(* CoDeSys 2.3 project: cy-12-wg-004.pro *)
(* Title: ClevergyAS - Albino E-02 *)
(* Version: 1.25 *)
(* Author: Andrea Ravasio *)
(* Libraries: Standard.lib 8.11.10 12:37:48, Util.lib 26.9.14 11:12:46, Visual.lib 8.11.10 12:37:48, Ethernet.lib 8.11.10 12:37:48, WagoLibIdent.lib 25.2.13 13:49:34, WagoLibMBX_01.lib 20.3.12 16:32:38, WagoLibStatus.lib 8.11.10 12:37:48, SysLibFile.lib 8.11.10 12:37:48, SysLibRtc.lib 8.11.10 12:37:48, SysLibSockets.lib 5.5.11 09:22:24, SysLibEvent.lib 8.11.10 12:37:48, SysLibPlcCtrl.lib 8.11.10 12:37:48, SysLibCallback.lib 8.11.10 12:37:48, ModbusEthernet_03.lib 15.5.15 16:47:39 *)

(* PLC configuration (modules and I/O channels)
VPN_ST1 AT %IX16.0 [BOOLOnX_I] Ch_1 Digital input
LAMP_AL AT %QX6.0 [BOOLOnX_Q] Ch_1 Digital output
KEY_QE_ST AT %IX16.1 [BOOLOnX_I] Ch_2 Digital input
CIR06_EN AT %QX6.1 [BOOLOnX_Q] Ch_2 Digital output
CIR07_AL AT %IX16.2 [BOOLOnX_I] Ch_3 Digital input
CIR05_EN AT %QX6.2 [BOOLOnX_Q] Ch_3 Digital output
CIR07_ST AT %IX16.3 [BOOLOnX_I] Ch_4 Digital input
CIR04_EN AT %QX6.3 [BOOLOnX_Q] Ch_4 Digital output
CIR07_AUT AT %IX16.4 [BOOLOnX_I] Ch_5 Digital input
CIR03_EN AT %QX6.4 [BOOLOnX_Q] Ch_5 Digital output
CIR06_AL AT %IX16.5 [BOOLOnX_I] Ch_6 Digital input
CIR02_EN AT %QX6.5 [BOOLOnX_Q] Ch_6 Digital output
CIR06_ST AT %IX16.6 [BOOLOnX_I] Ch_7 Digital input
CIR01_EN AT %QX6.6 [BOOLOnX_Q] Ch_7 Digital output
CIR06_AUT AT %IX16.7 [BOOLOnX_I] Ch_8 Digital input
CAL01_On_Off AT %QX6.7 [BOOLOnX_Q] Ch_8 Digital output
CIR05_AL AT %IX16.8 [BOOLOnX_I] Ch_1 Digital input
CIR07_EN AT %QX6.8 [BOOLOnX_Q] Ch_1 Digital output
CIR05_ST AT %IX16.9 [BOOLOnX_I] Ch_2 Digital input
CAL01_Rst_Bruc AT %QX6.9 [BOOLOnX_Q] Ch_2 Digital output
CIR05_AUT AT %IX16.10 [BOOLOnX_I] Ch_3 Digital input
AT %QX6.10 [BOOLOnX_Q] Ch_3 Digital output
CIR04_AL AT %IX16.11 [BOOLOnX_I] Ch_4 Digital input
AT %QX6.11 [BOOLOnX_Q] Ch_4 Digital output
CIR04_ST AT %IX16.12 [BOOLOnX_I] Ch_5 Digital input
AT %QX6.12 [BOOLOnX_Q] Ch_5 Digital output
CIR04_AUT AT %IX16.13 [BOOLOnX_I] Ch_6 Digital input
AT %QX6.13 [BOOLOnX_Q] Ch_6 Digital output
CIR03_AL AT %IX16.14 [BOOLOnX_I] Ch_7 Digital input
AT %QX6.14 [BOOLOnX_Q] Ch_7 Digital output
CIR03_ST AT %IX16.15 [BOOLOnX_I] Ch_8 Digital input
AT %QX6.15 [BOOLOnX_Q] Ch_8 Digital output
CIR03_AUT AT %IX17.0 [BOOLOnX_I] Ch_1 Digital input
CTL01_ST AT %IX17.1 [BOOLOnX_I] Ch_2 Digital input
CIR02_AUT AT %IX17.2 [BOOLOnX_I] Ch_3 Digital input
CIR01_AUT AT %IX17.3 [BOOLOnX_I] Ch_4 Digital input
ALARM_PM_PB_TB AT %IX17.4 [BOOLOnX_I] Ch_1 Digital input
CIR02_AL AT %IX17.5 [BOOLOnX_I] Ch_2 Digital input
UTA01_AL AT %IX17.6 [BOOLOnX_I] Ch_3 Digital input
CIR02_ST AT %IX17.7 [BOOLOnX_I] Ch_4 Digital input
CIR01_AL AT %IX17.8 [BOOLOnX_I] Ch_1 Digital input
CAL01_AL AT %IX17.9 [BOOLOnX_I] Ch_2 Digital input
CIR01_ST AT %IX17.10 [BOOLOnX_I] Ch_3 Digital input
CAL01_ManAuto AT %IX17.11 [BOOLOnX_I] Ch_4 Digital input
T_S01 AT %IW0 [INTOnW_I] Ch_1 signed Input value
T_S03 AT %IW1 [INTOnW_I] Ch_2 signed Input value
T_S02 AT %IW2 [INTOnW_I] Ch_3 signed Input value
T_S04 AT %IW3 [INTOnW_I] Ch_4 signed Input value
T_S05 AT %IW4 [INTOnW_I] Ch_1 signed Input value
T_S07 AT %IW5 [INTOnW_I] Ch_2 signed Input value
T_S06 AT %IW6 [INTOnW_I] Ch_3 signed Input value
AT %IW7 [INTOnW_I] Ch_4 signed Input value
T_S09 AT %IW8 [INTOnW_I] Ch_1 signed Input value
T_S08 AT %IW9 [INTOnW_I] Ch_2 signed Input value
AT %IW10 [INTOnW_I] Ch_3 signed Input value
AT %IW11 [INTOnW_I] Ch_4 signed Input value
VRD03_CTRL AT %QW0 [WORDOnW_Q] Ch_1 Analog output
VRD02_CTRL AT %QW1 [WORDOnW_Q] Ch_2 Analog output
VRD01_CTRL AT %QW2 [WORDOnW_Q] Ch_1 Analog output
VRD04_CTRL AT %QW3 [WORDOnW_Q] Ch_2 Analog output
CAL01_CRL AT %QW4 [WORDOnW_Q] Ch_1 Analog output
AT %QW5 [WORDOnW_Q] Ch_2 Analog output
VRD03_ST AT %IW12 [WORDOnW_I] Ch_1 Input word
VRD02_ST AT %IW13 [WORDOnW_I] Ch_2 Input word
0750-0478 2 AI 0-10V 16 Bit S.E. [Type_8_2_Channels] node 13, in %IB52 out %QB24 {INTTypePAAssignment = PLC; INTTypeModule = plugged}
  VRD01_ST AT %IW14 [WORDOnW_I] Ch_1 Input word
  VRD04_ST AT %IW15 [WORDOnW_I] Ch_2 Input word
0750-0513 2 DO 250V AC 2.0A Rel 2NO (PotFree) [Type_10_2_Channels] node 14, in %IB35 out %QB14 {INTTypePAAssignment = PLC; INTTypeModule = plugged}
  UTA_CTRL AT %QX7.0 [BOOLOnX_Q] Ch_1 Digital output
  AT %QX7.1 [BOOLOnX_Q] Ch_2 Digital output
Fieldbus variables [FB_VARS] node 1, in %IB0 out %QB0
Flag variables [FLAG_VARS] node 2, in %IB0 out %QB0
Modbus-Master [MB_MASTER] node 3, in %IB0 out %QB0
*)

(* Global variable list: Global_Constants *)
VAR_GLOBAL CONSTANT

	Plant_NAME			: STRING :='cySN:12 cyVER: E05 Palestra Centro Sportivo Rio Re ';
	Plant_SN			: DWORD  :=12;	(* S/N Impianto di telecontrollo *)
	Plant_SW_VER		: WORD   :=3;	(* Versione SW installata *)


	(* Parameters *)
	Plant_DefaultTAmb	: INT	:=100;		(* [.1°C] Temperatura ambiente di default in caso di rottura sonda *)
	Plant_MaxRunTAmb	: INT   :=250; 		(* [.1°C] Temperatura ambiente massima funzionamento impianto *)
	Plant_AntiFreezeTAmb: INT   :=-40;		(* [.1°C] Antifreeze temperature, start circulators *)
	Plant_CirOffDelay	: TIME	:=T#15m;	(* (Def.T#15m) Ritardo spegnimento pompe per ricircolo caldaia *)
	Plant_MaxWaterLoss	: WORD  :=2;		(* [lt/h] Massima perdita del circuito *)
	Plant_VRD_TDefault	: INT	:=300;		(* [.1°C] Temperatura di default in caso di errore climatica *)

	(* Filesystem *)
	FilesPath  			: STRING :='S:\';

(*	(* TCP Logger *)
	Logger_SERVER		: STRING:='';
	Logger_IP			: STRING:='192.168.100.3';
	Logger_PORT			: WORD  :=80;
	Logger_GETSTART		: STRING:='GET /cygmsrv/hsgm.ashx?';
	Logger_GETEND		: STRING:='$R$N$R$N';
	Logger_CHECK		: STRING:='True';
	Logger_CRLF			: STRING:='$R$N';
	Logger_DataFile		: STRING:='S:\LOG.DAT';
	Logger_DataFileOld	: STRING:='S:\LOG.BCK';
	Logger_IndexFile	: STRING:='S:\LOG.IDX';
	Logger_ConnRetries	: BYTE:=5;
	Logger_RecoverMsgs	: BYTE:=25;

	(* TCP Remote *)
	Remote_PORT			: WORD  :=10; (*44818; *)
	Remote_WELCOME		: STRING:='Connected$R$N';
	Remote_OK			: STRING:='OK$R$N';
	Remote_ERROR		: STRING:='ERROR$R$N';



	(* TCP Sockets *)
	MAX_SEND_TCP_SERVER					 : DWORD:=1500;(*60000*)
	MAX_RECEIVE_TCP_SERVER				 : DWORD:=3000;
	MAX_RECEIVE_TCP_SERVER_SOCKET	 	 : DWORD:=1500;
	MAX_SEND_TCP_CLIENT					 : DWORD:=3000;(*15000*)
	MAX_RECEIVE_TCP_CLIENT				 : DWORD:=1500;
	MAX_RECEIVE_TCP_CLIENT_SOCKET		 : DWORD:=1500;
	MAX_RECEIVE_UDP_SERVER				 : INT  :=1472;
	MAX_RECEIVE_UDP_CLIENT				 : INT  :=1472;
	CONNECT_WATCHDOG_TIME				 : TIME :=t#10s;
*)

	(* TCP Logger *)
	Logger_SERVER		: STRING:='';
	Logger_IP			: STRING:='192.168.100.3';
	Logger_PORT			: WORD  :=80;
	Logger_GETSTART		: STRING:='GET /cygmsrv/hsgm.ashx?';
	Logger_GETEND		: STRING:='$R$N$R$N';
	Logger_CHECK		: STRING:='True';
	Logger_CRLF			: STRING:='$R$N';
	Logger_DataFile		: STRING:='S:\LOG.DAT';
	Logger_DataFileOld	: STRING:='S:\LOG.BCK';
	Logger_IndexFile	: STRING:='S:\LOG.IDX';
	Logger_ConnRetries	: BYTE:=5;
	Logger_RecoverMsgs	: BYTE:=25;

	(* TCP Remote *)
	Remote_PORT			: WORD  :=10;
	Remote_WELCOME		: STRING:='Connected$R$N';
	Remote_OK			: STRING:='OK$R$N';
	Remote_ERROR		: STRING:='ERROR$R$N';

	(* TCP Sockets *)
	MAX_SEND_TCP_SERVER					 : DWORD:=3000;(*60000*)
	MAX_RECEIVE_TCP_SERVER				 : DWORD:=3000;
	MAX_RECEIVE_TCP_SERVER_SOCKET	 	 : DWORD:=1500;
	MAX_SEND_TCP_CLIENT					 : DWORD:=3000;(*15000*)
	MAX_RECEIVE_TCP_CLIENT				 : DWORD:=1500;
	MAX_RECEIVE_TCP_CLIENT_SOCKET		 : DWORD:=1500;
	MAX_RECEIVE_UDP_SERVER				 : INT  :=1472;
	MAX_RECEIVE_UDP_CLIENT				 : INT  :=1472;
	CONNECT_WATCHDOG_TIME				 : TIME :=t#10s;

	(* VISU COLORS *)
	COLOR_RED 			: DWORD:=16#2020F0;
	COLOR_YELLOW		: DWORD:=16#20F0F0;
	COLOR_GREEN			: DWORD:=16#20F020;
	COLOR_GREEN_OFF 	: DWORD:=16#006000;
	COLOR_LBLUE			: DWORD:=16#F0F080;
	COLOR_LIGHT_GREEN	: DWORD := 16#006000;





END_VAR

(* Global variable list: Global_Retain *)
VAR_GLOBAL RETAIN PERSISTENT
	CAL01_Clima : typ_Clima;
	VRD01_Clima : typ_Clima;
	VRD02_Clima : typ_Clima;
	VRD03_Clima : typ_Clima;
	VRD04_Clima : typ_Clima;

	CTL01_Count : DWORD;

	Mode_Manual : BOOL := FALSE;


	DelayAllarmeTemperaturaNonRaggiunta: INT;
	DeltaInterventoAllarmeTempeaturaNonRaggiuta: INT;
	OffsetSetPointManuale: INT;							(* Offset al Setpoint manuale per comensare lo scambiatore *)
	OffsetSetPointManuale2: INT;						(* Offset al Setpoint manuale per comensare lo scambiatore Aggiuntivo *)
	BitAbilitaBoost: BOOL:=TRUE;						(* Abilitiazione Boost *)
	RifOffsetBoost:INT;									(* Offset al Setpoint della Caldaia per azione di Boost *)

	SogliaMinStartAntigelo: INT;
	SogliaMinStopAntigelo: INT;
	BitAbilitaAntigelo: BOOL:=TRUE;


END_VAR

(* Global variable list: Global_Variables *)
VAR_GLOBAL

	SYS    : typ_SYS;
	Logger : typ_Logger;

	Lamp	:	LAMP_AL_GENERALE;

	T_AMB	:	INT;		(* Environment temperature *)


	(* Sonde Temperature impianto *)
	TPV01  : obj_TPV	:= ( ID:=1 ); 							   (* T_S01 Esterna *)
	TPV02  : obj_TPV	:= ( ID:=2 , IN_WMIN:=50 , IN_WMAX:=980 ); (* T_S02 Mandata Caldia *)
	TPV03  : obj_TPV	:= ( ID:=3 , IN_WMIN:=50 , IN_WMAX:=980 ); (* T_S03 Ritorno Caldaia *)
	TPV04  : obj_TPV	:= ( ID:=4 , IN_WMIN:=50 , IN_WMAX:=800 ); (* T_S04 FAN Coil Spogliatoio Piano Terra Radiatori*)
	TPV05  : obj_TPV	:= ( ID:=5 , IN_WMIN:=50 , IN_WMAX:=800 ); (* T_S05 Spogliatoio Primo Piano Radiatori *)
	TPV06  : obj_TPV	:= ( ID:=6 , IN_WMIN:=50 , IN_WMAX:=800 ); (* T_S06 Temperatura ACS *)
	TPV07  : obj_TPV	:= ( ID:=7 , IN_WMIN:=50 , IN_WMAX:=800 ); (* T_S07 Temperatura Bollitore *)
	TPV08  : obj_TPV	:= ( ID:=8 , IN_WMIN:=50 , IN_WMAX:=800 ); (* T_S08 Ingresso UTA *)
	TPV09  : obj_TPV	:= ( ID:=9 , IN_WMIN:=50 , IN_WMAX:=800 ); (* T_S09 Uscita UTA *)

	TAMB   : obj_TAMB	:= ( ID:=1 );
					(* vedi parametro G e Paramentro H manuale Caldaia UNICAL *)
	CAL01  : obj_CAL_01 := ( ID:=1,	LimiteMAXSetPoint:= 800,LimiteMinSetPoint:=300,OnDelay:=T#500ms,OffDelay:=T#500ms );


	(* Circolatori  *)
	CIR01  : obj_CIR_01 := ( ID:=1,CIR_AUTO:=TRUE, OnDelay:=T#1s, OffDelay:=T#5m);
	CIR02  : obj_CIR_01 := ( ID:=2,CIR_AUTO:=TRUE, OnDelay:=T#2s, OffDelay:=T#1s); (* Controllo Palestra UTA *)
	CIR03  : obj_CIR_01 := ( ID:=3,CIR_AUTO:=TRUE, OnDelay:=T#3s, OffDelay:=T#1s); (* Controllo Palestra Piano Terra Radiatori *)
	CIR04  : obj_CIR_01 := ( ID:=4,CIR_AUTO:=TRUE, OnDelay:=T#4s, OffDelay:=T#1s); (* Controllo Spogliatoi Primo Piano Radiatori *)
	CIR05  : obj_CIR_01 := ( ID:=5,CIR_AUTO:=TRUE, OnDelay:=T#5s, OffDelay:=T#1s); (* Controllo Circolatore Bollitore  *)
	CIR06  : obj_CIR_01 := ( ID:=6,CIR_AUTO:=TRUE, OnDelay:=T#6s, OffDelay:=T#1s); (* Controllo Circolatore Bollitore  *)
	CIR07  : obj_CIR_01 := ( ID:=7,CIR_AUTO:=TRUE, OnDelay:=T#7s, OffDelay:=T#1s); (* Controllo Circolatore ACS *)


	(* Valvole motorizzate Analogiche  *)
	VRD01	:	obj_VRD_02:= (ID:=1, fFeedback:=TRUE, ReducedRange := FALSE,Local_VRD_TAlarm:=800); (* Controllo Palestra Piano Terra Radiatori *)
	VRD02	:	obj_VRD_02:= (ID:=2, fFeedback:=TRUE, ReducedRange := FALSE,Local_VRD_TAlarm:=800); (* Controllo Spogliatoi Primo Piano Radiatori *)
(* VRD03 Esclusa perchè bypassata *)
(*	VRD03	:	obj_VRD_02:= (ID:=3, fFeedback:=TRUE, ReducedRange := FALSE,Local_VRD_TAlarm:=800); (* Controllo Circolatore Bollitore  *) *)
	VRD04	:	obj_VRD_02:= (ID:=4, fFeedback:=TRUE, ReducedRange := FALSE,Local_VRD_TAlarm:=800); (* Controllo Palestra UTA *)


	(* Crono termostati *)
	THER01 : obj_CRONTER := ( ID:=1, Local_MaxRunTAmb:=800,Histeresys:=10); (* Controllo Palestra UTA *)
	THER02 : obj_CRONTER := ( ID:=2, Local_MaxRunTAmb:=800,Histeresys:=10);	(* Controllo Palestra Piano Terra Radiatori *)
	THER03 : obj_CRONTER := ( ID:=3, Local_MaxRunTAmb:=800,Histeresys:=10);	(* Controllo Spogliatoi Primo Piano Radiatori *)
	THER04 : obj_CRONTER := ( ID:=4, Local_MaxRunTAmb:=800,Histeresys:=50);	(* Controllo Circolatore Bollitore  *)
	THER05 : obj_CRONTER := ( ID:=5, Local_MaxRunTAmb:=800,Histeresys:=10);	(* Controllo Circolatore ACS *)
	THER250: obj_CRONTER := ( ID:=250, Local_MaxRunTAmb:=800,Histeresys:=10);(* Controllo Boost *)

	CronEd : obj_CRON_EDITOR;

	(* Contalitri *)
	CTL01	:	obj_CTL	:= (ID:=1, Peso:=10);
	UTA01  : obj_UTA:=(ID:=1);



	UTA01_ST: BOOL;
	UTA01_Antigelo: BOOL;
	UTA01_ManAut: BOOL;
END_VAR

(* Data type in LON/Enumerations *)
TYPE alarm_type_t :
(
	AL_HEADER := -13,
	AL_FOOTER := -12,
	AL_DEBUG := -11,
	AL_INFO := -10,
	AL_SYSTEM_INFO := -6,
	AL_VALUE_INVALID := -5,
	AL_CONSTANT := -4,
	AL_OFFLINE := -3,
	AL_UNKNOWN := -2,
	AL_NUL := -1,
	AL_NO_CONDITION := 0,
	AL_ALM_CONDITION := 1,
	AL_TOT_SVC_ALM_1 := 2,
	AL_TOT_SVC_ALM_2 := 3,
	AL_TOT_SVC_ALM_3 := 4,
	AL_LOW_LMT_CLR_1 := 5,
	AL_LOW_LMT_CLR_2 := 6,
	AL_HIGH_LMT_CLR_1 := 7,
	AL_HIGH_LMT_CLR_2 := 8,
	AL_LOW_LMT_ALM_1 := 9,
	AL_LOW_LMT_ALM_2 := 10,
	AL_HIGH_LMT_ALM_1 := 11,
	AL_HIGH_LMT_ALM_2 := 12,
	AL_FIR_ALM := 13,
	AL_FIR_PRE_ALM := 14,
	AL_FIR_TRBL := 15,
	AL_FIR_SUPV := 16,
	AL_FIR_TEST_ALM := 17,
	AL_FIR_TEST_PRE_ALM := 18,
	AL_FIR_ENVCOMP_MAX := 19,
	AL_FIR_MONITOR_COND := 20,
	AL_FIR_MAINT_ALERT := 21,
	AL_FATAL_ERROR := 30,
	AL_ERROR := 31,
	AL_WARNING := 32
);
END_TYPE

(* Data type in Errors *)
TYPE en_Logger_ErrLev :
(
	EL_Log			:=0,
	EL_Wrn			:=1,
	EL_Alarm		:=2,
	EL_AlarmStop	:=3
);
END_TYPE

(* Data type in Errors *)
TYPE en_Logger_Status :
(
	S_Logger_UNKNOWN := 0,
	S_Logger_IDLE,
	S_Logger_WAITCONN,
	S_Logger_WAITTX,
	S_Logger_WAITRESP,
	S_Logger_ERROR
);
END_TYPE

(* Data type *)
TYPE en_SYS_Objects :
(
	EO_SYS		:=0,  (* PLC *)
	EO_VPN		:=1,  (* VPN *)
	EO_DOOR		:=2,  (* Door & access control *)

	EO_CAL		:=10, (* Caldaia *)
	EO_CIR		:=11, (* Circolatore *)
	EO_CRON		:=12, (* Crono-termostato *)
	EO_VRD		:=13, (* Valvola miscelatore pannelli *)
	EO_CTL		:=14, (* Contalitri *)
	EO_CTB		:=15, (* Contabilizzatore *)
	EO_TPV		:=16, (* Temperature probes values *)
	EO_PPV		:=17, (* Pressure probes values *)
	EO_PBV		:=18, (* Over-Pressure Alarms *)
	EO_TBV		:=19, (* Over-Temperature Alarms *)
	EO_PMV		:=20, (* Under-Pressure Alarms *)
	EO_GRU		:=21, (* Gruppo termico *)
	EO_PDC		:=22, (* Pompa di calore *)
	EO_SOL		:=23, (* Pannello solare termico *)
	EO_ESOL		:=24, (* Pannello solare fotovoltaico *)
	EO_GAS		:=25, (* Contatore GAS *)
	EO_PORT		:=26, (* Misuratore di portata *)
	EO_FPV		:=27, (* Flow probes values *)
	EO_ANZ		:=28, (* Analizzatore di rete *)
	EO_SCA		:=29, (* Signal Control Alarms *)
	EO_LUX		:=30, (* Base Illumination point *)
	EO_LUXM		:=31, (* Metered Illumination point *)
	EO_PSG		:=32, (* Sensore di passaggio *)
	EO_HVAC		:=33, (* Heating, Ventilating and Air Conditioning *)
	EO_HYGRV	:=34, (* Relative Humidity sensors value *)
	EO_COOV		:=35, (* Carbon Dioxide CO2 sensors value *)
	EO_INV		:=36, (* Inverter *)
	EO_STR		:=37, (* Smart string box *)

	EO_CIRD		:=39, (* Double CIR *)
	EO_ACS		:=40, (* Hot domestic water *)
	EO_FRG		:=41, (* Frigo *)
	EO_THER		:=42, (* Thermostat *)
	EO_CIRM		:=43, (* Modbus CIR *)
	EO_CIRDM	:=44, (* Modbus double CIR *)
	EO_UTA		:=47, (* Modbus double CIR *)

	EO_ZGW			:=200,  (* ZigBee - Gateway *)
	EO_ZRM			:=201,	(* ZigBee - Repeater *)
	EO_ZREL			:=202,	(* ZigBee - Actuator rele *)
	EO_ZTHL			:=203,	(* ZigBee - Temperature Sensor *)

	EO_ASGW			:=250,	(* ASi - Gateway *)
	EO_ASCBI		:=251,	(* ASi - Input Board, Ciabatta *)

	EO_LON			:=1000, (* Bus - LON *)
	EO_MODBUS		:=1001, (* Bus - MODBUS *)
	EO_MBUS			:=1002, (* Bus - M-BUS *)
	EO_MODBUS_TCP	:=1003, (* Bus - MODBUS TCP *)

	EO_GENERIC		:=9000, (* Generic dataset *)
	EO_EXPO			:=9001 (* EXPO dataset *)
);
END_TYPE

(* Data type *)
TYPE en_SYS_Status :
(
	S_UNKNOWN  := 0,
	S_STARTUP,
	S_INIT_RTC,
	S_INIT_VAR,
	S_AUTOTEST,
	S_RUNNING,
	S_SHUTDOWN,
	S_HALT
);
END_TYPE

(* Data type in LON/Enumerations *)
TYPE file_request_t :
(
	FR_NUL := -1,
	FR_OPEN_TO_SEND := 0,
	FR_OPEN_TO_RECEIVE := 1,
	FR_CLOSE_FILE := 2,
	FR_CLOSE_DELETE_FILE := 3,
	FR_DIRECTORY_LOOKUP := 4,
	FR_OPEN_TO_SEND_RA := 5,
	FR_OPEN_TO_RECEIVE_RA := 6
);
END_TYPE

(* Data type in LON/Enumerations *)
TYPE file_status_t :
(
	FS_NUL := -1,
	FS_XFER_OK := 0,
	FS_LOOKUP_OK := 1,
	FS_OPEN_FAIL := 2,
	FS_LOOKUP_ERR := 3,
	FS_XFER_UNDERWAY := 4,
	FS_IO_ERR := 5,
	FS_TIMEOUT_ERR := 6,
	FS_WINDOW_ERR := 7,
	FS_AUTH_ERR := 8,
	FS_ACCESS_UNAVAIL := 9,
	FS_SEEK_INVALID := 10,
	FS_SEEK_WAIT := 11
);
END_TYPE

(* Data type in LON/Enumerations *)
TYPE hvac_t :
(
	HVAC_NUL := -1,
	HVAC_AUTO := 0,
	HVAC_HEAT := 1,
	HVAC_MRNG_WRMUP := 2,
	HVAC_COOL := 3,
	HVAC_NIGHT_PURGE := 4,
	HVAC_PRE_COOL := 5,
	HVAC_OFF := 6,
	HVAC_TEST := 7,
	HVAC_EMERG_HEAT := 8,
	HVAC_FAN_ONLY := 9,
	HVAC_FREE_COOL := 10,
	HVAC_ICE := 11,
	HVAC_MAX_HEAT := 12,
	HVAC_ECONOMY := 13,
	HVAC_DEHUMID := 14,
	HVAC_CALIBRATE := 15,
	HVAC_EMERG_COOL := 16,
	HVAC_EMERG_STEAM := 17,
	HVAC_MAX_COOL := 18,
	HVAC_HVC_LOAD := 19,
	HVAC_NO_LOAD := 20
);
END_TYPE

(* Data type in LON/Enumerations *)
TYPE object_request_t :
(
	RQ_NUL := -1,
	RQ_NORMAL := 0,
	RQ_DISABLED := 1,
	RQ_UPDATE_STATUS := 2,
	RQ_SELF_TEST := 3,
	RQ_UPDATE_ALARM := 4,
	RQ_REPORT_MASK := 5,
	RQ_OVERRIDE := 6,
	RQ_ENABLE := 7,
	RQ_RMV_OVERRIDE := 8,
	RQ_CLEAR_STATUS := 9,
	RQ_CLEAR_ALARM := 10,
	RQ_ALARM_NOTIFY_ENABLED := 11,
	RQ_ALARM_NOTIFY_DISABLED := 12,
	RQ_MANUAL_CTRL := 13,
	RQ_REMOTE_CTRL := 14,
	RQ_PROGRAM := 15,
	RQ_CLEAR_RESET := 16,
	RQ_RESET := 17,
	RQ_CLEAR_LOG := 18,
	RQ_LOAD_PROGRAM := 19,
	RQ_RUN_PROGRAM := 20,
	RQ_HALT_PROGRAM := 21,
	RQ_RESTART_PROGRAM := 22,
	RQ_UNLOAD_PROGRAM := 23,
	RQ_STEP_PROGRAM := 24
);
END_TYPE

(* Data type in LON/Enumerations *)
TYPE priority_level_t :
(
	PR_NUL := -1,
	PR_LEVEL_0 := 0,
	PR_LEVEL_1 := 1,
	PR_LEVEL_2 := 2,
	PR_LEVEL_3 := 3,
	PR_1 := 4,
	PR_2 := 5,
	PR_3 := 6,
	PR_4 := 7,
	PR_6 := 8,
	PR_8 := 9,
	PR_10 := 10,
	PR_16 := 11
);
END_TYPE

(* Data type in Plant_Objects *)
TYPE typ_Clima : (* CURVA CLIMATICA *)
STRUCT
	InitOK:		BOOL;
	Points: 	ARRAY [0..10] OF POINT;
END_STRUCT
END_TYPE

(* Data type in Plant_Objects *)
TYPE typ_Cron_Calendar :
STRUCT
	Profile		: ARRAY[0..384] OF BYTE;
END_STRUCT
END_TYPE

(* Data type in Plant_Objects *)
TYPE typ_Cron_Jolly :
STRUCT
	Start		: DT;
	End			: DT;
	Temp		: WORD;
	Flags		: WORD; (* B0:Enabled B1..B15:Unused *)
END_STRUCT
END_TYPE

(* Data type in Plant_Objects *)
TYPE typ_Cron_Profile :
STRUCT
	Flags		: WORD;
	Setpoint	: ARRAY [0..95] OF WORD;
END_STRUCT
END_TYPE

(* Data type in Errors *)
TYPE typ_Logger :
STRUCT
	Status		: en_Logger_Status;

	SendReq		: BOOL;
	SendIdx		: DWORD;
	SendData	: ARRAY [0..MAX_SEND_TCP_CLIENT] OF BYTE;
	SendLen		: DINT;

	TData		: ARRAY [0..MAX_SEND_TCP_CLIENT] OF BYTE;
	TLen		: DINT;

	LastIdxPos	: DWORD;

	(* Temporary variables used by objects *)
	s1			: STRING(256);
	i1			: WORD;


END_STRUCT
END_TYPE

(* Data type in Plant_Objects *)
TYPE typ_MODBUS_VAR : (* Gestione parametri MODBUS *)
STRUCT
	SlaveAddress	: BYTE;
	FunCode			: BYTE;
	FunAddress		: WORD;
	Refresh_Time	: BYTE; (* 0:No refresh x:Refresh in seconds *)
	Refresh_Cnt		: BYTE; (* INTERNAL *)
	Variable		: POINTER TO WORD;
	Variable_Size	: BYTE;
	Variable_Mirror : WORD; (* INTERNAL [Force refresh on read variables when <>0] *)
END_STRUCT
END_TYPE

(* Data type *)
TYPE typ_SYS :
STRUCT
	Status			: en_SYS_Status;
	Warning			: BOOL;
	Alarm			: BOOL;
	AlarmStop		: BOOL;

	Time_LogString	: STRING;
	Time_Year		: WORD;
	Time_Month		: BYTE;
	Time_Day		: BYTE;

	Time_CT_DT		: DT;
	Time_CT_Day		: WORD;
	Time_CT_Quarter	: BYTE;

	LastLogs_Idx	: BYTE;
	LastLogs_Dat	: ARRAY[0..5] OF STRING;
	LastLogs_Msg	: ARRAY[0..5] OF STRING;

END_STRUCT
END_TYPE

(* Data type in LON/NetworkVariables *)
TYPE typSnvtAlarm : 
STRUCT
	abLocation : ARRAY[0..5] OF BYTE;
	wObjectId : WORD;
	bAlarmType : BYTE (* enum type alarm_type_t *);
	bPriorityLevel : BYTE (* enum type priority_level_t *);
	wIndexToSnvt : WORD;
	abValue : ARRAY[0..3] OF BYTE;
	wYear : WORD;
	bMonth : BYTE;
	bDay : BYTE;
	bHour : BYTE;
	bMinute : BYTE;
	bSecond : BYTE;
	wMillisecond : WORD;
	abAlarmLimit : ARRAY[0..3] OF BYTE;
	bStatusInformation : BYTE; (* bit allocation of bStatusInformation:
	bit 0: NVI update counter LSB
	bit 1: NVI update counter
	bit 2: NVI update counter
	bit 3: NVI update counter MSB
	bit 4: timeout for NVI occurs (MaxRcvTime expired)
	bit 5: reserved
	bit 6: reserved
	bit 7: force NVO update *)
	bInternalUseOnly : BYTE; (* Do not use this byte in your application! *)
END_STRUCT
END_TYPE

(* Data type in LON/NetworkVariables *)
TYPE typSnvtFilePos : 
STRUCT
	diRwPtr : DINT;
	wRwLength : WORD;
	bStatusInformation : BYTE; (* bit allocation of bStatusInformation:
	bit 0: NVI update counter LSB
	bit 1: NVI update counter
	bit 2: NVI update counter
	bit 3: NVI update counter MSB
	bit 4: timeout for NVI occurs (MaxRcvTime expired)
	bit 5: reserved
	bit 6: reserved
	bit 7: force NVO update *)
	bInternalUseOnly : BYTE; (* Do not use this byte in your application! *)
END_STRUCT
END_TYPE

(* Data type in LON/NetworkVariables *)
TYPE typSnvtFileReq : 
STRUCT
	bRequest : BYTE (* enum type file_request_t *);
	wIndex : WORD;
	wReceiveTimeout : WORD;
	abDestAddress : ARRAY[0..4] OF BYTE (* union declaration *);
	bAuthOn : BYTE;
	bPrioOn : BYTE;
	bStatusInformation : BYTE; (* bit allocation of bStatusInformation:
	bit 0: NVI update counter LSB
	bit 1: NVI update counter
	bit 2: NVI update counter
	bit 3: NVI update counter MSB
	bit 4: timeout for NVI occurs (MaxRcvTime expired)
	bit 5: reserved
	bit 6: reserved
	bit 7: force NVO update *)
	bInternalUseOnly : BYTE; (* Do not use this byte in your application! *)
END_STRUCT
END_TYPE

(* Data type in LON/NetworkVariables *)
TYPE typSnvtFileStatus : 
STRUCT
	bStatus : BYTE (* enum type file_status_t *);
	wNumberOfFiles : WORD;
	wSelectedFile : WORD;
	abAdr : ARRAY[0..21] OF BYTE (* union declaration *);
	bStatusInformation : BYTE; (* bit allocation of bStatusInformation:
	bit 0: NVI update counter LSB
	bit 1: NVI update counter
	bit 2: NVI update counter
	bit 3: NVI update counter MSB
	bit 4: timeout for NVI occurs (MaxRcvTime expired)
	bit 5: reserved
	bit 6: reserved
	bit 7: force NVO update *)
	bInternalUseOnly : BYTE; (* Do not use this byte in your application! *)
END_STRUCT
END_TYPE

(* Data type in LON/NetworkVariables *)
TYPE typSnvtHvacMode : 
STRUCT
	bSnvtHvacMode : BYTE (* enum type hvac_t *);
	bStatusInformation : BYTE; (* bit allocation of bStatusInformation:
	bit 0: NVI update counter LSB
	bit 1: NVI update counter
	bit 2: NVI update counter
	bit 3: NVI update counter MSB
	bit 4: timeout for NVI occurs (MaxRcvTime expired)
	bit 5: reserved
	bit 6: reserved
	bit 7: force NVO update *)
	bInternalUseOnly : BYTE; (* Do not use this byte in your application! *)
END_STRUCT
END_TYPE

(* Data type in LON/NetworkVariables *)
TYPE typSnvtObjRequest : 
STRUCT
	wObjectId : WORD;
	bObjectRequest : BYTE (* enum type object_request_t *);
	bStatusInformation : BYTE; (* bit allocation of bStatusInformation:
	bit 0: NVI update counter LSB
	bit 1: NVI update counter
	bit 2: NVI update counter
	bit 3: NVI update counter MSB
	bit 4: timeout for NVI occurs (MaxRcvTime expired)
	bit 5: reserved
	bit 6: reserved
	bit 7: force NVO update *)
	bInternalUseOnly : BYTE; (* Do not use this byte in your application! *)
END_STRUCT
END_TYPE

(* Data type in LON/NetworkVariables *)
TYPE typSnvtObjStatus : 
STRUCT
	wObjectId : WORD;
	bBitfieldByteOffset2 : BYTE (* bit field *);
	bBitfieldByteOffset3 : BYTE (* bit field *);
	bBitfieldByteOffset4 : BYTE (* bit field *);
	bBitfieldByteOffset5 : BYTE (* bit field *);
	bStatusInformation : BYTE; (* bit allocation of bStatusInformation:
	bit 0: NVI update counter LSB
	bit 1: NVI update counter
	bit 2: NVI update counter
	bit 3: NVI update counter MSB
	bit 4: timeout for NVI occurs (MaxRcvTime expired)
	bit 5: reserved
	bit 6: reserved
	bit 7: force NVO update *)
	bInternalUseOnly : BYTE; (* Do not use this byte in your application! *)
END_STRUCT
END_TYPE

(* Data type in LON/NetworkVariables *)
TYPE typSnvtState : 
STRUCT
	bBitfieldByteOffset0 : BYTE (* bit field *);
	bBitfieldByteOffset1 : BYTE (* bit field *);
	bStatusInformation : BYTE; (* bit allocation of bStatusInformation:
	bit 0: NVI update counter LSB
	bit 1: NVI update counter
	bit 2: NVI update counter
	bit 3: NVI update counter MSB
	bit 4: timeout for NVI occurs (MaxRcvTime expired)
	bit 5: reserved
	bit 6: reserved
	bit 7: force NVO update *)
	bInternalUseOnly : BYTE; (* Do not use this byte in your application! *)
END_STRUCT
END_TYPE

(* Data type in LON/NetworkVariables *)
TYPE typSnvtSwitch : 
STRUCT
	bValue : BYTE;
	siState : SINT;
	bStatusInformation : BYTE; (* bit allocation of bStatusInformation:
	bit 0: NVI update counter LSB
	bit 1: NVI update counter
	bit 2: NVI update counter
	bit 3: NVI update counter MSB
	bit 4: timeout for NVI occurs (MaxRcvTime expired)
	bit 5: reserved
	bit 6: reserved
	bit 7: force NVO update *)
	bInternalUseOnly : BYTE; (* Do not use this byte in your application! *)
END_STRUCT
END_TYPE

(* Data type in LON/NetworkVariables *)
TYPE typSnvtTempP :
STRUCT
	iSnvtTempP : INT;
	bStatusInformation : BYTE; (* bit allocation of bStatusInformation:
	bit 0: NVI update counter LSB
	bit 1: NVI update counter
	bit 2: NVI update counter
	bit 3: NVI update counter MSB
	bit 4: timeout for NVI occurs (MaxRcvTime expired)
	bit 5: reserved
	bit 6: reserved
	bit 7: force NVO update *)
	bInternalUseOnly : BYTE; (* Do not use this byte in your application! *)
END_STRUCT
END_TYPE

(* Data type in LON/NetworkVariables *)
TYPE typSnvtTimeStamp : 
STRUCT
	iYear : INT;
	bMonth : BYTE;
	bDay : BYTE;
	bHour : BYTE;
	bMinute : BYTE;
	bSecond : BYTE;
	bStatusInformation : BYTE; (* bit allocation of bStatusInformation:
	bit 0: NVI update counter LSB
	bit 1: NVI update counter
	bit 2: NVI update counter
	bit 3: NVI update counter MSB
	bit 4: timeout for NVI occurs (MaxRcvTime expired)
	bit 5: reserved
	bit 6: reserved
	bit 7: force NVO update *)
	bInternalUseOnly : BYTE; (* Do not use this byte in your application! *)
END_STRUCT
END_TYPE

(* POU PLC_PRG, ST *)
PROGRAM PLC_PRG
VAR
	Timer1: TON; (* Fast controls tick *)
	Timer2: TON; (* Plant control tick *)
	Timer3: TON; (* Logger timer *)

	SecCircuitLogic	:	BOOL;	(* Secondary circuit request: LOGICAL ON/OFF *)
	SecCircuitReal	:	BOOL;	(* Secondart circuit request: REAL ON/OFF	 *)




	StartCAL_Antigelo: RS;
	fAntigelo		:FLT_TAP;  (* Sgnalazione LOG Antigelo  *)


	OffsetBoost: INT;
	pippo: WORD;
	HMI_AggiornaLog: BOOL;
	SetPointVRD04: INT;

	OffsetVRD04: INT;

END_VAR

VAR RETAIN
	HMISetPointVRD04: INT;
	HMI_LimitMaxOut: INT;
	HMI_LimitMinOut:INT;
	HMI_LimitMinIN: INT;
	HMI_LimitMaxIN: INT;
END_VAR
(******************************************************************************
 ****                           MAIN TASK CODE                             ****
 ******************************************************************************

	Network setup:
		IP  = 192.168.100.2 | MSK = 255.255.255.0
		GW	= 192.168.100.1 | DNS = 192.168.100.1
		SNTP = 193.204.114.232 (3600s) ==> 192.168.100.3
*)

(*==============================*)
(*===== Main status machine ====*)
(*==============================*)
Main_Stm();

(*==============================*)
(*== Running cycle operations ==*)
(*==============================*)
(*
IF SYS.Status>S_INIT_VAR THEN

	(* Update LON output variables (needs to be here to obtain only one refresh) *)
	CAL01.Heartbeat( CLIM:=CAL01_Clima );
	(* Execute LON process *)
	Module_1_PRG();

END_IF
*)
(*==============================*)
(*== System cycle operations ===*)
(*==============================*)
(* Execute TCP processes *)
Logger_Proc();
Remote_Proc();
(* Update user led *)
USRLED_Update();
(* Execute Cron Editor commands *)
CronEd();
END_PROGRAM
ACTION Main_Stm:
CASE Sys.Status OF

	S_STARTUP:
		Sys.Status:=S_INIT_RTC;

	S_INIT_RTC:
		(* Check RTC and update from network *)
		RTC_Update();
		(* Check time *)
		IF Sys.Time_Year>2000 THEN
			Sys.Status:=S_INIT_VAR;
		END_IF








	S_INIT_VAR:
		LogEv(EL_Wrn,EO_SYS,0,1,CONCAT('System_startup_v',WORD_TO_STRING(Plant_SW_VER)));
		Sys.Status:=S_RUNNING;

	S_RUNNING:
		Timer1(IN:=NOT Timer1.Q,PT:=T#50ms);
		IF Timer1.Q THEN
			(* Update meters *)
			CTL01 ( CTL_ST:=CTL01_ST, COUNT:=CTL01_Count );
			(* Update system checks *)
			SYS_Proc();
		END_IF

		Timer2(IN:=NOT Timer2.Q,PT:=T#500ms);
		IF Timer2.Q THEN
			(* Read current date/time *)
			RTC_Update();
			(* Execute plant operations *)
			TPV01	 ( IN:=T_S01);
			TPV02	 ( IN:=T_S02);
			TPV03	 ( IN:=T_S03);
			TPV04	 ( IN:=T_S04);
			TPV05	 ( IN:=T_S05);
			TPV06	 ( IN:=T_S06);
			TPV07	 ( IN:=T_S07);
			TPV08	 ( IN:=T_S08);
			TPV09	 ( IN:=T_S09);

		(*	TAMB  ( IN1:=TPV01.IN ); *)
			T_AMB:=TPV01.IN;

			(* Crono, CronoTermostati e boost ed eventuale Antigelo  *)

(*
		  (* Gestione Ciclo antigelo : in questo impianto il ciclo antigelo è gestito coi crono ambiente *)

			StartCAL_Antigelo(	SET:=(SogliaMinStartAntigelo>TPV03.AVG),
								RESET1:= (TPV03.AVG>SogliaMinStopAntigelo) OR NOT BitAbilitaAntigelo
							);



			fAntigelo(IN:=StartCAL_Antigelo.Q1);
			IF fAntigelo.EVH THEN
				LogEv(EL_Log,EO_SYS,0,11,'Ciclo_Antigelo_Attivato');
			END_IF
			IF fAntigelo.EVL THEN
				LogEv(EL_Log,EO_SYS,0,12,'Ciclo_Antigelo_Disattivato');
			END_IF
*)



			THER01();						(* gestito solo Crono *)
			CIR02.OnOff:=THER01.RunCrono; 	(* UTA Palestra Fan Coil *) (* OR StartCAL_Antigelo.Q1 -- per introdurre start antigelo *)

			THER02();						(* gestito solo Crono *)
			CIR03.OnOff:=THER02.RunCrono; 	(* Spogliatoio Piano Terra Radiatori *)

			THER03();						(* gestito solo Crono *)
			CIR04.OnOff:=THER03.RunCrono; 	(* Spgliatoio Piano Primo Radiatori *)

			THER04(Temperature:=TPV07.IN);				(* gestito solo Cronotermostato *)
			CIR05.OnOff:=CIR06.OnOff:=THER04.Run; 	(* Bollitore *)

			THER05();						(* gestito solo Crono *)
			CIR07.OnOff:=THER05.RunCrono; 	(* Lancio ACS *)

			(* il crono virtuale 250 è quello che gestisce il boost.
				 Questo è attivo se da remoto lo abilitano ed è subordinato alla verifica della Temperatura 
				imposta nel Crono con quella di una data temperatura *)
			THER250();						(* Boost *)
			RifOffsetBoost:=LIMIT(0,RifOffsetBoost,200);
			OffsetBoost:=SEL(BitAbilitaBoost,0,SEL((THER250.SetPoint>TPV08.AVG),0,RifOffsetBoost));


			(* VRD *)
			(*  l'offset Boost viene fatto direttamente sulle cliamtiche delle VRD perchè nonesiste la curva cliamtica della caldaia *)
			VRD01(TempControlloCC:=T_AMB,
					RUN:=CIR03.Run,
					CLIM:=VRD01_Clima,
					OffsetBoost:=OffsetBoost,
					TEMP:=TPV04.IN,
					STATUS:=VRD01_ST,
					OUT=>VRD01_CTRL);

			VRD02(TempControlloCC:=T_AMB,
					RUN:=CIR04.Run,
					CLIM:=VRD02_Clima,
					OffsetBoost:=OffsetBoost,
					TEMP:=TPV05.IN,
					STATUS:=VRD02_ST,
					OUT=>VRD02_CTRL);

			(* in questo caso la VRD03 è bypassata sempre al 100% *)

(*			VRD03( RUN:=CIR05.Pump_ST ,
					ComandoManuale:=TRUE ,
					RiferimentoManuale:=100 ,
					CLIM:=VRD03_Clima,
					OffsetBoost:=OffsetBoost,
					TEMP:=0,(*TPV07.AVG,*)
					STATUS:=VRD03_CTRL, (*VRD03_ST,*)
					OUT=>VRD03_CTRL) ; (*VRD03_CTRL); *)
*)

(* Controllo Set Point Valvola VRD 04:
				- La Temperatura di ritorno dell'Aria TS08 fornirà il riferimento alla Curva CLiamtica alla Caldaia  
				- La Variabile di Processo della VRD sarà la temperatura di Mandata dell'aria TS09. Il Set Pont sarà un valore
				  fisso impostabiledal WebVisu e saà corretto se la temperatura TS08 aumenterà troppo con un caurva linearizzata
				  sempre impostavile da WebVisu



*)




			OffsetVRD04:=LINEAR_BAD(
									PuntoMinX:=HMI_LimitMinOut,
									PuntoMaxX:=HMI_LimitMaxOut,
									ValIn:=TPV08.AVG,
									PuntoMinY:=HMI_LimitMinIN,
									PuntoMaxY:=HMI_LimitMaxIN,
									Decimali:=0);

			OffsetVRD04:=LIMIT(HMI_LimitMinOut,OffsetVRD04,HMI_LimitMaxOut);

			SetPointVRD04:=HMISetPointVRD04 - OffsetVRD04;




			VRD04(	TempControlloCC:=TPV08.AVG,
					AbilitaSetPointManuale:=TRUE,
					SetPointManuale:=SetPointVRD04,
					RUN:=UTA01.Run,
					ComandoManuale:=NOT THER04.Run ,
					RiferimentoManuale:=100 ,
					CLIM:=VRD04_Clima,
					OffsetBoost:=OffsetBoost,
					TEMP:=TPV08.AVG,
					STATUS:=VRD04_ST,
					OUT=>VRD04_CTRL);


			(* Gestione Caldaia *)

			(* Secondary circuit heat request *)
			SecCircuitLogic := 	CIR02.Ctrl_Run
								OR CIR03.Ctrl_Run
								OR CIR04.Ctrl_Run
								OR (CIR05.Ctrl_Run AND CIR06.Ctrl_Run )
								;
			SecCircuitReal := 	CIR02.Run
								OR CIR03.Run
								OR CIR04.Run
								OR (CIR05.Run AND CIR06.Run )
								;
			(* Circolatore primario Caldaia *)
			CIR01.OnOff := SEL(SecCircuitLogic,FALSE,TRUE) AND SYS.AlarmStop=FALSE;


			(* Gestione Caldaia *)
			CAL01.Run := CIR01.Run ;

			(* Scrivo il setpoint in funzione della curva cliamatica più alta *)

			(* Set Point Caldaia *)

			CAL01.SetPointManuale:=CAL01.Curve_Temp - OffsetSetPointManuale + OffsetBoost;  	(* Temperaratura del Boost *)
			CAL01.SetPointManuale:=MAX(CAL01.SetPointManuale,SEL(CIR06.OnOff,0,THER04.SetPoint  + OffsetSetPointManuale2)); (* Bollitore *)
			CAL01.SetPointManuale:=MAX(CAL01.SetPointManuale,SEL(VRD01.RUN,0,VRD01.Ctrl_SetPoint ));
			CAL01.SetPointManuale:=MAX(CAL01.SetPointManuale,SEL(VRD02.RUN,0,VRD02.Ctrl_SetPoint ));
			CAL01.SetPointManuale:=MAX(CAL01.SetPointManuale,SEL(VRD04.RUN,0,VRD04.Ctrl_SetPoint ));


			(* VRD03 Esclusa perchè bypassata *)

			 (* la scelta del set point è dinamica quindi  bisogna settare il bit in AbilitaSetPointManuale perchhè
				non viene preso in automatico nel blocco CAL *)
			CAL01(CLIM:=CAL01_Clima,AbilitaSetPointManuale:=TRUE);




			(* Gestione Circolatori *)

			CIR01 ( Pump_AL:=NOT CIR01_AL , Pump_ST:=CIR01_ST ,Pump_AUTO:=CIR01_AUT, CIR_EN=>CIR01_EN );
			CIR02 ( Pump_AL:=NOT CIR02_AL , Pump_ST:=CIR02_ST ,Pump_AUTO:=CIR02_AUT, CIR_EN=>CIR02_EN );
			CIR03 ( Pump_AL:=NOT CIR03_AL , Pump_ST:=CIR03_ST ,Pump_AUTO:=CIR03_AUT,CIR_EN=>CIR03_EN );
			CIR04 ( Pump_AL:=NOT CIR04_AL , Pump_ST:=CIR04_ST ,Pump_AUTO:=CIR04_AUT,CIR_EN=>CIR04_EN );
			CIR05 ( Pump_AL:=NOT CIR05_AL , Pump_ST:=CIR05_ST ,Pump_AUTO:=CIR05_AUT,CIR_EN=>CIR05_EN );
			CIR06 ( Pump_AL:=NOT CIR06_AL , Pump_ST:=CIR06_ST ,Pump_AUTO:=CIR06_AUT, CIR_EN=>CIR06_EN );
			CIR07 ( Pump_AL:=NOT CIR07_AL , Pump_ST:=CIR07_ST ,Pump_AUTO:=CIR07_AUT,CIR_EN=>CIR07_EN );




			UTA01(RUN:=THER01.RunCrono,
					UTA_CentrAL:= UTA01_AL,
					DO_OUT=>UTA_CTRL);


			VRD01 ( CLIM:=VRD01_Clima , TEMP:=TPV04.IN , STATUS:=VRD01_ST , RUN:=CIR03_EN ,	OUT=>VRD01_CTRL );
			VRD02 ( CLIM:=VRD02_Clima , TEMP:=TPV05.IN , STATUS:=VRD02_ST , RUN:=CIR04_EN ,	OUT=>VRD02_CTRL );
(* VRD03 Esclusa perchè bypassata *)
(*			VRD03 ( CLIM:=VRD03_Clima , TEMP:=TPV06.IN , STATUS:=VRD02_ST , RUN:=CIR07_EN ,	OUT=>VRD03_CTRL );*)
			VRD04 ( CLIM:=VRD04_Clima , TEMP:=TPV08.IN , STATUS:=VRD04_ST , RUN:=CIR02_EN ,	OUT=>VRD04_CTRL );



			CAL01(AI_Potenza:= CAL01_CRL,
					CAL_ST:=CAL01_On_Off,
					ALARM_CAL:= CAL01_AL ,
					PresenzaFiamma:=CAL01_On_Off,
					CmdCALAuto_MAN:= NOT CAL01_ManAuto,
					CLIM:=CAL01_Clima ,
					AO_SetPoint=>CAL01_CRL ,
					CAL_EN=>CAL01_On_Off  ,
					DO_RIARMO=>CAL01_Rst_Bruc ,
					 );


					(* RUN:=( CIR02.Run OR CIR03.Run  OR CIR04.Run  OR  CIR05.Run OR  CIR06.Run)			(* RUN Caldaia *)
										AND SYS.AlarmStop=FALSE
										AND ALARM_PM_PB_TB	(**** Allarme ISPESL ****)
										AND CIR01.Status_Log=0

										 ); *)

			Lamp( Allarme:=	CAL01.Status_Log=2 OR
  						  	CIR01.Status_Log=2 OR
  						  	CIR02.Status_Log=2 OR
  						  	CIR03.Status_Log=2 OR
 						  	CIR04.Status_Log=2 OR
						  	CIR05.Status_Log=2 OR
						  	CIR06.Status_Log=2 OR
						  	CIR07.Status_Log=2 OR
							TPV01.Status_Log=2 OR
							TPV02.Status_Log=2 OR
							TPV03.Status_Log=2 OR
							TPV04.Status_Log=2 OR
							TPV05.Status_Log=2 OR
							TPV06.Status_Log=2 OR
							TPV07.Status_Log=2 OR
							TPV08.Status_Log=2 OR
							TPV09.Status_Log=2 OR
							THER01.Status_Log=2 OR
							THER02.Status_Log=2 OR
							THER03.Status_Log=2 OR
							THER04.Status_Log=2 OR
							THER05.Status_Log=2 OR
							THER250.Status_Log=2 OR
							VRD01.Status_Log=2 OR
							VRD02.Status_Log=2 OR
(* VRD03 Esclusa perchè bypassata *)
(*							VRD03.Status_Log=2 OR*)
							VRD04.Status_Log=2 OR
							UTA01.Status_Log=2
							,
							Warning:=	CAL01.Status_Log=1 OR
  						  	CIR01.Status_Log=1 OR
  						  	CIR02.Status_Log=1 OR
  						  	CIR03.Status_Log=1 OR
 						  	CIR04.Status_Log=1 OR
						  	CIR05.Status_Log=1 OR
						  	CIR06.Status_Log=1 OR
						  	CIR07.Status_Log=1 OR
							TPV01.Status_Log=1 OR
							TPV02.Status_Log=1 OR
							TPV03.Status_Log=1 OR
							TPV04.Status_Log=1 OR
							TPV05.Status_Log=1 OR
							TPV06.Status_Log=1 OR
							TPV07.Status_Log=1 OR
							TPV08.Status_Log=1 OR
							TPV09.Status_Log=1 OR
							THER01.Status_Log=1 OR
							THER02.Status_Log=1 OR
							THER03.Status_Log=1 OR
							THER04.Status_Log=1 OR
							THER05.Status_Log=1 OR
							THER250.Status_Log=1 OR
							VRD01.Status_Log=1 OR
							VRD02.Status_Log=1 OR
(* VRD03 Esclusa perchè bypassata *)
(*							VRD03.Status_Log=1 OR *)
							VRD04.Status_Log=1 OR
							UTA01.Status_Log=1
							,
							AllarmeLampada=>LAMP_AL
							);


			(* Test toggle *)
		(*	IF TEST1 THEN TEST1:=FALSE; ELSE TEST1:=TRUE; END_IF*)
		END_IF

		Timer3(IN:=NOT Timer3.Q,PT:=T#5m);
		IF Timer3.Q OR HMI_AggiornaLog THEN
			(* Trig logger *)
			LogTrig();
			(* Execute temporary CSV logger *)
			CSV_Log();
		END_IF

	S_SHUTDOWN:
		(* Stop caldaia *)
		(* Stop deviatori *)
		(* Aspetta 5 min prima di spegnere eventuali circolatori *)
		Sys.Status:=S_STARTUP;

	S_HALT:
		(* Aspetta uscita manuale *)
		Sys.Status:=S_STARTUP;


ELSE
	Sys.Status:=S_STARTUP;
END_CASE;
END_ACTION

(* POU Utils Functions/FLT_TAP, ST *)
FUNCTION_BLOCK FLT_TAP
VAR_INPUT
	IN		: BOOL;
	TAP		: BYTE:=4;
	INITEV	: BOOL:=TRUE;
END_VAR
VAR_OUTPUT
	OUT		: BOOL;
	EVH		: BOOL;
	EVL		: BOOL;
END_VAR
VAR
	init	: BOOL:=FALSE;
	cnt		: BYTE;
END_VAR
EVH:=FALSE;
EVL:=FALSE;

IF NOT init THEN
	init := TRUE;
	IF INITEV THEN
		OUT  := NOT IN;
		cnt  := TAP;
	ELSE
		OUT  := IN;
	END_IF
END_IF

IF OUT<>IN THEN
	cnt:=cnt+1;
	IF cnt>TAP THEN
		OUT:=IN;
		cnt:=0;
		IF OUT THEN EVH:=TRUE; ELSE EVL:=TRUE; END_IF
	END_IF
ELSE
	cnt:=0;
END_IF
END_FUNCTION_BLOCK

(* POU TCP_Logger/Logger_Proc, ST *)
PROGRAM Logger_Proc
VAR
	c1:         	TCPCLIENT;

	Open:	    	BOOL;
	IpAddr:			DWORD;
	InetAddr:		DWORD;
	Connected:  	BOOL;
	Error:      	DINT;
	TxTrig:     	BOOL;
	RxData:			ARRAY [0..MAX_RECEIVE_TCP_CLIENT] OF BYTE;
	RxLen:			DINT;

	Retry:			BYTE;	(* Counter for connection retries *)
	Recovered:		BYTE;	(* Counter for recovered unsent messages *)

	i:				DINT;
	pos:			DWORD;
	hFile:			DWORD;

END_VAR
(*=== State machine ===*)
CASE Logger.Status OF

	S_Logger_UNKNOWN:
		(* Startup *)
		Logger.SendReq:=FALSE;
		Open:=FALSE;
		Logger.Status:=S_Logger_IDLE;

	S_Logger_IDLE:
		(* Wait request *)
		IF Logger.SendReq THEN
			(* Resolve server name or use static IP *)
			IF LEN(Logger_SERVER)=0 THEN
				InetAddr:=SysSockInetAddr(Logger_IP);
			ELSE
				IpAddr:=SysSockGetHostByName(ADR(Logger_SERVER));
				DWORDSWAP(pIn:=ADR(IpAddr), pOut:=ADR(InetAddr));
			END_IF
			TxTrig:=FALSE;
			RxLen:=0;
			(* Open connection *)
			Open:=TRUE;
			Logger.Status:=S_Logger_WAITCONN;
		END_IF

	S_Logger_WAITCONN:
		(* Wait connection *)
		IF Connected THEN
			(* Send data *)
			TxTrig:=TRUE;
			Logger.Status:=S_Logger_WAITTX;
		END_IF
		IF Error>0 THEN
			Open:=FALSE;
			Logger.Status:=S_Logger_ERROR;
		END_IF

	S_Logger_WAITTX:
		(* Wait transmission *)
		IF NOT TxTrig THEN
			Logger.Status:=S_Logger_WAITRESP;
		END_IF
		IF Error>0 THEN
			Open:=FALSE;
			Logger.Status:=S_Logger_ERROR;
		END_IF

	S_Logger_WAITRESP:
		(* Wait response *)
		IF Connected=FALSE (* OR TIMEOUT!! *) THEN
			Open:=FALSE;
			(* Check response *)
			IF RxLen>=4 AND CHKSTRING(pString:=ADR(RxData), pPattern:=ADR(Logger_CHECK)) THEN
				Logger.SendReq:=FALSE;
				Retry:=0;
				(* Check unsent messages to flush *)
				IF Recovered<Logger_RecoverMsgs THEN
					MsgChk();
					IF Logger.SendReq=TRUE THEN
						Recovered:=Recovered+1;
					ELSE
						Recovered:=0;
					END_IF
				ELSE
					Recovered:=0;
				END_IF
				Logger.Status:=S_Logger_IDLE;
			ELSE
				Logger.Status:=S_Logger_ERROR;
			END_IF
		END_IF

	S_Logger_ERROR:
		(* Connection error or send failure *)
		Retry:=Retry+1;
		IF Retry>Logger_ConnRetries THEN
			(* Save message as unsent *)
			MsgSave();
			Logger.SendReq:=FALSE;
			Retry:=0;
		END_IF
		Logger.Status:=S_Logger_IDLE;

ELSE
	Logger.Status:=S_Logger_UNKNOWN;
END_CASE


(*=== Execute client lib ===*)
c1(
	xOpenConnection			:= Open,
	dwInetAddr 				:= InetAddr,
	wPortNumber				:= Logger_PORT,
	ptSendData				:= ADR(Logger.SendData),
	diSendCount				:= Logger.SendLen,
	tConnectWatchdogTime	:= t#10s,
	xStartSend				:= TxTrig,
	aReceiveBuffer			:= RxData,
	diReceiveCount			:= RxLen,
	xConnected				=> Connected,
	diError					=> Error
);

(*=== Process Rx data ===*)
(*IF RxLen>0 THEN
	RxLen:=0;
END_IF*)
END_PROGRAM
ACTION MsgChk:
(* Open index file *)
hFile:=SysFileOpen(Logger_IndexFile,'r');
IF hFile=0 THEN
	RETURN;
END_IF
(* Search oldest message to recover *)
SysFileSetPos(hFile,Logger.LastIdxPos);
Logger.SendLen:=0;
REPEAT
	SysFileRead(hFile, ADR(Logger.SendIdx), SIZEOF(Logger.SendIdx));
	pos:=SysFileGetPos(hFile);
	SysFileRead(hFile, ADR(Logger.SendLen), SIZEOF(Logger.SendLen));
UNTIL
	SysFileEOF(hFile) OR Logger.SendLen<>0
END_REPEAT
SysFileClose(hFile);
(* Delete index file when all messages are recovered *)
IF Logger.SendLen=0 THEN
	Logger.LastIdxPos:=0;
	SysFileDelete(Logger_IndexFile);
	RETURN;
END_IF
(* Recover message data *)
hFile:=SysFileOpen(Logger_DataFile,'r');
IF hFile<>0 THEN
	SysFileSetPos(hFile,Logger.SendIdx);
	SysFileRead(hFile,ADR(Logger.SendData),Logger.SendLen);
	Logger.SendReq:=TRUE;
	SysFileClose(hFile);
END_IF
(* Clear index entry *)
hFile:=SysFileOpen(Logger_IndexFile,'a');
IF hFile<>0 THEN
	SysFileSetPos(hFile,pos);
	i:=0;
	SysFileWrite(hFile, ADR(i), 4);
	Logger.LastIdxPos:=SysFileGetPos(hFile);
	SysFileClose(hFile);
END_IF
END_ACTION
ACTION MsgSave:
(* Add log position in recovery indexes *)
hFile:=SysFileOpen(Logger_IndexFile,'a');
SysFileWrite(hFile, ADR(Logger.SendIdx), SIZEOF(Logger.SendIdx));
SysFileWrite(hFile, ADR(Logger.SendLen), SIZEOF(Logger.SendLen));
SysFileClose(hFile);
END_ACTION

(* POU Utils Functions/TCPCLIENT, ST *)
FUNCTION_BLOCK TCPCLIENT
(***********************************************************************************************************	*)
(* Version: 1.3b                        			          													*)
(* Date: 28.10.2014                   				          							            			*)
(***********************************************************************************************************	*)
(* WAGO Kontakttechnik GmbH Hansastr. 27 32423 Minden(Westf.)													*)
(* Tel. +0049 571/887-0 Fax. +0049 571/887-0																	*)
(* Author: VB																									*)
(***********************************************************************************************************	*)
(*Description:	A TCP client to read and write data with additional connection watchdog							*)
(*History:																										*)
(*Version 1.3b: 28.10.2014: Use DWORD address for IP (Andrea Ravasio)											*)
(*Version 1.3: 11.02.2011: Changes according to 750-880/881											 			*)
(*Version 1.2: 29.08.2007 Bugfix TCP Client																		*)
(*Version 1.1: 15.01.2007 Changes according to FW11																*)
(*Version 1.0: 09.03.2006 Release																				*)
(***********************************************************************************************************	*)
VAR CONSTANT
	STATE_CREATE     				 : BYTE:= 0;
	STATE_OPEN     					 : BYTE:= 1;
	STATE_IOCTL    					 : BYTE:= 2;
	STATE_CONNECT     				 : BYTE:= 10;
	STATE_TX       					 : BYTE:= 20;
	STATE_RX       					 : BYTE:= 30;
	STATE_CLOSE    					 : BYTE:= 40;
	STATE_ERROR_TRAP			     : BYTE:= 200;
END_VAR

VAR_INPUT
	xOpenConnection					: BOOL;
	dwInetAddr						: DWORD; (* <== Use SysSockInetAddr() value or
													swapped bytes order of SysSockGetHostByName() value *)
	wPortNumber						: WORD;
	ptSendData						: POINTER TO ARRAY[0..MAX_SEND_TCP_CLIENT] OF BYTE;
	diSendCount						: DINT;
	tConnectWatchdogTime		    : TIME := t#10s;
END_VAR
VAR_OUTPUT
	xConnected						: BOOL;
	diError 						: DINT := 0;
END_VAR
(* ErrorCodes -----------------------------------------
	16#8001 => No socket descriptor available 
	16#8002 => SysSockSend returns -1 
	16#8003 => Socket was "gracefully closed" 
	16#8004 => switching to none blocking mode fails
	16#8005 => SysSockClose() returns FALSE 
    16#8006 => SysSockConnect() fails
    16#8007 => SysSockSend() fails
	16#8008 => error state machine 
	16#8009 => timeout while waiting for data from server 
------------------------------------------------------------*)
VAR_IN_OUT
	xStartSend							: BOOL;
	aReceiveBuffer						: ARRAY [0..MAX_RECEIVE_TCP_CLIENT] OF BYTE;
	diReceiveCount						: DINT;
END_VAR
VAR
	m_State								: BYTE := 0;
	m_ReceiveBuffer						: ARRAY [0..MAX_RECEIVE_TCP_CLIENT_SOCKET] OF BYTE;
	m_Socket							: DINT;
	m_AddressInfo						: SOCKADDRESS;
	m_BytesReceived						: DINT;
	m_diReturn							: DINT;
	m_xReturn							: BOOL;
	m_IoCtlParameter  					: DINT := 1; (* IOCTL-Parameter for non-blocking mode of sockets *)
	i									: INT;
	T_Connect							: TON;
	m_count								: DINT;
	diOption							: DINT := 1;
	m_Blocking   						: DINT := 0;
END_VAR
IF xOpenConnection THEN
	(* State maschine *)
	CASE  m_State OF

	(* -------------------------------------------------------------------------*)
	STATE_CREATE:
			(* create socket descriptor*)
			m_Socket := SysSockCreate(diAddressFamily	:= SOCKET_AF_INET,
													 diType		:= SOCKET_STREAM,
													 diProtocol := SOCKET_IPPROTO_TCP);
			IF m_Socket >= 0 THEN
			(*Set Push-Bit*)
				IF ADR(%MW0)=16#30000000  OR ADR(%MW0)=16#20000000 THEN (*841 or 881*)
					SysSockSetOption(
						diSocket:=m_Socket,
						diLevel:=6,
						diOption:=SOCKET_TCP_NODELAY,
						pOptionValue:=ADR(diOption),
						diOptionLength:=SIZEOF(diOption));
				ELSE
						;
				END_IF
				m_State := STATE_IOCTL; (* succesful *)
			ELSE
				diError := 16#8001;  (* no socket descriptor available *)
				m_State := STATE_ERROR_TRAP;
			END_IF

	(* -------------------------------------------------------------------------*)
	STATE_IOCTL: (* change  socket mode  to none blocking *)
		m_diReturn := SysSockIoctl( m_Socket, SOCKET_FIONBIO, ADR(m_IoCtlParameter));
		IF m_diReturn <> 0 THEN
			m_AddressInfo.sin_family := SOCKET_AF_INET;
			m_AddressInfo.sin_port := SysSockNtohs(wPortNumber);
			m_AddressInfo.sin_addr := dwInetAddr;
			m_State := STATE_CONNECT;
		ELSE
			diError := 16#8004;  (* switching to none blocking mode fails *)
			m_State := STATE_ERROR_TRAP;
		END_IF


	(* -------------------------------------------------------------------------*)
	STATE_CONNECT: (* connect with server *)
		T_Connect(IN:=TRUE , PT:=tConnectWatchdogTime);(*activate watchdog for establishing connection to a server*)
		m_xReturn := SysSockConnect ( m_Socket, ADR(m_AddressInfo),  SIZEOF(m_AddressInfo));
		IF m_xReturn THEN (* succesful *)
			IF xStartSend THEN
				m_State := STATE_TX;(*transmit data*)
			ELSE
				m_State := STATE_RX;(*wait for data from server*)
			END_IF
			xConnected:=TRUE;
			T_Connect(IN:=FALSE);
		ELSE
			IF T_Connect.Q THEN
				diError := 16#8006;  (* connect fails *)
				xConnected:=FALSE;
				T_Connect(IN:=FALSE);
				m_State := STATE_ERROR_TRAP;
				SysSockClose( m_Socket);
			ELSE
				m_State := STATE_CONNECT;(*client still  tries to set up connection*)
			END_IF
		END_IF


	STATE_TX:	 (* send TCP-message *)
		m_diReturn := SysSockSend(diSocket := m_Socket,
								  pbyBuffer := ADR(ptSendData^[0]),
								  diBufferSize := diSendCount-m_count,
								  diFlags := 0);

		CASE m_diReturn OF
		-1:	(* ERROR *)
			T_Connect(IN:=TRUE , PT:=CONNECT_WATCHDOG_TIME);(*activate watchdog to check communication*)
			IF t_Connect.Q THEN
				diError := 16#8007;
				T_Connect(IN:=FALSE);
				m_State:=STATE_CLOSE;
			END_IF
		0: (* socket was "gracefully closed" *)
			m_State := STATE_CLOSE;
			diError := 16#8003;
		ELSE (* succesful *)
			m_count:=m_count+m_diReturn;
			IF m_count>=diSendCount THEN
				diError := 16#0000;
				m_State := STATE_RX;
				m_count:=0;
				xStartSend:=FALSE;
			END_IF
			T_Connect(IN:=FALSE);
		END_CASE

	(* -------------------------------------------------------------------------*)
	STATE_RX: (* process receive data *)
			m_BytesReceived := SysSockRecv(	diSocket 	:= m_Socket,
										pbyBuffer 	:= ADR(m_ReceiveBuffer),		(* Address of receive buffer *)
										diBufferSize:= SIZEOF(m_ReceiveBuffer),
										diFlags		:= 0);

			CASE m_BytesReceived OF
			-1:	(* No data available or error occured *)
				T_Connect(IN:=TRUE , PT:=tConnectWatchdogTime);(*activate watchdog to check communication*)
				IF t_Connect.Q THEN
					diError:=16#8009;
					T_Connect(IN:=FALSE);
					m_State:=STATE_CLOSE;
				END_IF
				IF xStartSend THEN
					m_State:=STATE_TX	;(* WAIT IN THIS STATE  and check for arriving data or new send command*)
				END_IF;
			0: (* socket was "gracefully closed"  *)
				m_State:=STATE_CLOSE;
				diError := 16#8003;
			ELSE (* succesful *)
				diError := 16#0000;
				T_Connect(IN:=FALSE);
				(* Copy received data into receive buffer *)
				FOR i:= 0 TO DINT_TO_INT(m_BytesReceived	)-1 DO
					aReceiveBuffer[diReceiveCount]:= m_ReceiveBuffer[i];
					diReceiveCount:=(diReceiveCount+1) MOD SIZEOF(aReceiveBuffer);
				END_FOR

			END_CASE

	(* -------------------------------------------------------------------------*)
	STATE_CLOSE : (* close socket *)
		IF ADR(%MW0)=16#30000000  OR ADR(%MW0)=16#20000000 THEN (*841 or 881*)
			;
		ELSE
			SysSockShutdown(m_Socket, 0);;(*870*)
		END_IF
		m_xReturn := SysSockClose( m_Socket);
		m_Socket := -1;
		m_State := 0; (* succesful *)
		xConnected:=FALSE;
		T_Connect(IN:=FALSE);
	(* -------------------------------------------------------------------------*)
	STATE_ERROR_TRAP: (* error handling *)
		xConnected:=FALSE;

	ELSE  (* Bad FSM code trap  *)
			m_State:= STATE_ERROR_TRAP;
			diError:= 16#8008;
	END_CASE

ELSE(*close connection*)
	IF m_Socket >= 0 THEN
		IF ADR(%MW0)=16#30000000  OR ADR(%MW0)=16#20000000 THEN (*841 or 881*)
			;
		ELSE
			SysSockShutdown(m_Socket, 0);;(*870*)
		END_IF
		SysSockClose( m_Socket);
	END_IF
	m_Socket := -1;
	diError := 16#0000;
	m_State := STATE_CREATE;
	xConnected:=FALSE;
	T_Connect(IN:=FALSE);
END_IF
END_FUNCTION_BLOCK

(* POU Utils Functions/DWORDSWAP, ST *)
FUNCTION DWORDSWAP:BOOL
VAR_INPUT
	pIn:POINTER TO ARRAY[1..4] OF BYTE;
	pOut:POINTER TO ARRAY[1..4] OF BYTE;
END_VAR
VAR
END_VAR
pOut^[1]:=pIn^[4];
pOut^[2]:=pIn^[3];
pOut^[3]:=pIn^[2];
pOut^[4]:=pIn^[1];
END_FUNCTION

(* POU Utils Functions/CHKSTRING, ST *)
FUNCTION CHKSTRING : BOOL
VAR_INPUT
	pString: POINTER TO BYTE;
	pPattern: POINTER TO BYTE;
END_VAR
VAR
END_VAR
CHKSTRING:=TRUE;
WHILE pPattern^<>0 AND CHKSTRING DO
	IF pPattern^<>pString^ THEN CHKSTRING:=FALSE; END_IF
	pString:=pString+1;
	pPattern:=pPattern+1;
END_WHILE
END_FUNCTION

(* POU TCP_Remote/Remote_Proc, ST *)
PROGRAM Remote_Proc
VAR
	s1:         	TCPSERVER;
	Enable: 		BOOL;
	Connected: 		BOOL;
	Error: 			DINT;

	TxData:			ARRAY[0..MAX_SEND_TCP_SERVER] OF BYTE;
	TxLen:			DINT;
	TxTrig:			BOOL;

	RxData:			ARRAY [0..MAX_RECEIVE_TCP_SERVER] OF BYTE;
	RxLen:			DINT;

	Status:			DINT;

	(* Command interpreter *)

	Cmd_Buf:		ARRAY [0..MAX_RECEIVE_TCP_SERVER] OF BYTE;
	Cmd_Buf_U16:	POINTER TO WORD;
	Cmd_Buf_INT:	POINTER TO INT;
	Cmd_BufLen:		WORD;
	Cmd_St:			WORD;

	Cmd_Obj:		WORD;
	Cmd_ObjIdx:		WORD;
	Cmd_C:			WORD;
	Cmd_R:			WORD;
	Cmd_CLen:		WORD;
	Cmd_RLen:		WORD;

	i : WORD;
	j : INT;


		(* per aggiornare la data e l'ora *)
	SetAnno: INT;
	SetMese: INT;
	SetGiorno: INT;
	SetOra: INT;
	SetMinuti: INT;
	SetSecondi: INT;


END_VAR
(*=== State machine ===*)
CASE Status OF
	0: (* Startup *)
		TxLen:=0; TxTrig:=FALSE;
		RxLen:=0;
		Enable:=TRUE;
		Status:=1;

	1: (* Wait incoming connection *)
		IF Connected THEN
			(* Log access *)
			LogEv(EL_Log,EO_VPN,1,5,'Remote');
			(* Send welcome message *)
			(*ADDSTRING(pTxData:=ADR(TxData), pString:=ADR(Remote_WELCOME), TxLen:=TxLen);
			TxTrig:=TRUE;*)
			Cmd_BufLen:=0;
			Cmd_St:=0;
			Status:=2;
		END_IF
		IF Error>1 THEN
			Enable:=FALSE;
			Status:=0;
		END_IF

	2: (* Wait command *)
		IF RxLen>0 THEN
			(*=== Interpreter start ===*)
			IF Cmd_BufLen+(RxLen/2)>=MAX_RECEIVE_TCP_SERVER THEN
				(* ERROR *)
				Cmd_BufLen:=0;
			ELSE
				i:=HEXTORAW(pString:=ADR(RxData), StringLen:=DINT_TO_WORD(RxLen), pData:=ADR(Cmd_Buf[Cmd_BufLen]));
				Cmd_BufLen:=Cmd_BufLen+i;
			END_IF
			IF Cmd_BufLen>=8 THEN
				Cmd_Buf_U16:=ADR(Cmd_Buf[6]);
				IF Cmd_BufLen>=(8+Cmd_Buf_U16^) THEN
					Cmd_CLen:=Cmd_Buf_U16^;
					Cmd_Buf_U16:=ADR(Cmd_Buf[0]); Cmd_Obj:=Cmd_Buf_U16^;
					Cmd_Buf_U16:=ADR(Cmd_Buf[2]); Cmd_ObjIdx:=Cmd_Buf_U16^;
					Cmd_Buf_U16:=ADR(Cmd_Buf[4]); Cmd_C:=Cmd_Buf_U16^;
					Command();
					Cmd_BufLen:=0;
				END_IF
			END_IF
			(*=== Interpreter end ===*)
			RxLen:=0;
		END_IF
		IF NOT Connected THEN
			Status:=0;
		END_IF

ELSE
	Status:=0;
END_CASE


(*=== Execute server lib ===*)
s1(
	xEnable				:= Enable,
	wPortNumber			:= Remote_PORT,
	tServerTimeOut		:= t#15m,
	ptSendData			:= ADR(TxData),
	diSendCount			:= TxLen,
	xStartSend			:= TxTrig,
	aReceiveBuffer		:= RxData,
	diReceiveCount		:= RxLen,
	xClientConnected	=> Connected,
	diError				=> Error
);
END_PROGRAM
ACTION Cmd_CAL:
(* Check index *)
IF Cmd_ObjIdx<>1 THEN
	Cmd_R:=2;
	RETURN;
END_IF

(* Process command *)
CASE Cmd_C OF

	1: (* GET CLIMATIC *)
		Cmd_RLen:=20;
		FOR i:=0 TO 4 DO
			j:=DINT_TO_INT(CAL01_Clima.Points[i].X);
			TxLen:=TxLen+RAWTOHEX(ADR(j),2,ADR(TxData[TxLen]));
			j:=DINT_TO_INT(CAL01_Clima.Points[i].Y);
			TxLen:=TxLen+RAWTOHEX(ADR(j),2,ADR(TxData[TxLen]));
		END_FOR

	2: (* SET CLIMATIC *)
		IF Cmd_CLen<>20 THEN
			Cmd_R:=4;
		ELSE
			FOR i:=0 TO 4 DO
				Cmd_Buf_INT:=ADR(Cmd_Buf[8+4*i]); j:=Cmd_Buf_INT^;
				CAL01_Clima.Points[i].X:=INT_TO_DINT(j);
				Cmd_Buf_INT:=ADR(Cmd_Buf[10+4*i]); j:=Cmd_Buf_INT^;
				CAL01_Clima.Points[i].Y:=INT_TO_DINT(j);
			END_FOR
		END_IF

	3: (* SET RESET *)

			CAL01.Rearm :=TRUE;

	4: (* SET Tempi delay On Off Ccaldaia  *)
		CASE Cmd_ObjIdx OF
			1:	Cmd_Buf_U16:=ADR(Cmd_Buf[8]);
				CAL01.OnDelay := DWORD_TO_TIME((Cmd_Buf_U16^)*60*1000); 			(* Delay ON*)
				Cmd_Buf_U16:=ADR(Cmd_Buf[10]);
				CAL01.OffDelay := DWORD_TO_TIME((Cmd_Buf_U16^)*60*1000);			(* Delay OFF *)

		END_CASE


	5: (* GET Tempi delay On Off Caldaia *)
		Cmd_RLen:=4;

			CASE Cmd_ObjIdx OF

			1:	j:=DWORD_TO_WORD(TIME_TO_DWORD((CAL01.OnDelay)/60/1000));
				TxLen:=TxLen+RAWTOHEX(ADR(j),2,ADR(TxData[TxLen]));
				j:=DWORD_TO_WORD(TIME_TO_DWORD((CAL01.OffDelay)/60/1000));
				TxLen:=TxLen+RAWTOHEX(ADR(j),2,ADR(TxData[TxLen]));
		END_CASE

ELSE
	Cmd_R:=3;
END_CASE
END_ACTION
ACTION Cmd_CIR:
IF Cmd_ObjIdx<1 OR Cmd_ObjIdx>6 THEN
	Cmd_R:=2;
	RETURN;
END_IF

(* Process command *)
CASE Cmd_C OF

	1:	(* Force CIR On *)
		CASE Cmd_ObjIdx OF

			1:	CIR01.CIR_RUN_REQ := TRUE;
			2:	CIR02.CIR_RUN_REQ := TRUE;
			3:	CIR03.CIR_RUN_REQ := TRUE;
			4:	CIR04.CIR_RUN_REQ := TRUE;
			5:	CIR05.CIR_RUN_REQ := TRUE;
			6:	CIR06.CIR_RUN_REQ := TRUE;
			7:	CIR07.CIR_RUN_REQ := TRUE;

		END_CASE

	2:	(* Force CIR Off *)
		CASE Cmd_ObjIdx OF

			1:	CIR01.CIR_STOP_REQ := TRUE;
			2:	CIR02.CIR_STOP_REQ := TRUE;
			3:	CIR03.CIR_STOP_REQ := TRUE;
			4:	CIR04.CIR_STOP_REQ := TRUE;
			5:	CIR05.CIR_STOP_REQ := TRUE;
			6:	CIR06.CIR_STOP_REQ := TRUE;
			7:	CIR07.CIR_STOP_REQ := TRUE;

		END_CASE

	3:	(* Release force *)
		CASE Cmd_ObjIdx OF

			1:	CIR01.CIR_RUN_REQ	:= FALSE;
				CIR01.CIR_STOP_REQ 	:= FALSE;
			2:	CIR02.CIR_RUN_REQ	:= FALSE;
				CIR02.CIR_STOP_REQ 	:= FALSE;
			3:	CIR03.CIR_RUN_REQ	:= FALSE;
				CIR03.CIR_STOP_REQ 	:= FALSE;
			4:	CIR04.CIR_RUN_REQ	:= FALSE;
				CIR04.CIR_STOP_REQ 	:= FALSE;
			5:	CIR05.CIR_RUN_REQ	:= FALSE;
				CIR05.CIR_STOP_REQ 	:= FALSE;
			6:	CIR06.CIR_RUN_REQ	:= FALSE;
				CIR06.CIR_STOP_REQ 	:= FALSE;
			7:	CIR07.CIR_RUN_REQ	:= FALSE;
				CIR07.CIR_STOP_REQ 	:= FALSE;

		END_CASE

	4: (* SET Tempi delay On Off Circolatori  *)
		CASE Cmd_ObjIdx OF
			1:	Cmd_Buf_U16:=ADR(Cmd_Buf[8]);
				CIR01.OnDelay := DWORD_TO_TIME((Cmd_Buf_U16^)*60*1000); 			(* Delay ON*)
				Cmd_Buf_U16:=ADR(Cmd_Buf[10]);
				CIR01.OffDelay := DWORD_TO_TIME((Cmd_Buf_U16^)*60*1000);			(* Delay OFF *)
			2:	Cmd_Buf_U16:=ADR(Cmd_Buf[8]);
				CIR02.OnDelay := DWORD_TO_TIME((Cmd_Buf_U16^)*60*1000);			(* Delay ON*)
				Cmd_Buf_U16:=ADR(Cmd_Buf[10]);
				CIR02.OffDelay := DWORD_TO_TIME((Cmd_Buf_U16^)*60*1000);			(* Delay OFF *)
			3:	Cmd_Buf_U16:=ADR(Cmd_Buf[8]);
				CIR03.OnDelay := DWORD_TO_TIME((Cmd_Buf_U16^)*60*1000);			(* Delay ON*)
				Cmd_Buf_U16:=ADR(Cmd_Buf[10]);
				CIR03.OffDelay := DWORD_TO_TIME((Cmd_Buf_U16^)*60*1000);			(* Delay OFF *)
			4:	Cmd_Buf_U16:=ADR(Cmd_Buf[8]);
				CIR04.OnDelay := DWORD_TO_TIME((Cmd_Buf_U16^)*60*1000);			(* Delay ON*)
				Cmd_Buf_U16:=ADR(Cmd_Buf[10]);
				CIR04.OffDelay := DWORD_TO_TIME((Cmd_Buf_U16^)*60*1000);			(* Delay OFF *)
			5:	Cmd_Buf_U16:=ADR(Cmd_Buf[8]);
				CIR05.OnDelay := DWORD_TO_TIME((Cmd_Buf_U16^)*60*1000);			(* Delay ON*)
				Cmd_Buf_U16:=ADR(Cmd_Buf[10]);
				CIR05.OffDelay := DWORD_TO_TIME((Cmd_Buf_U16^)*60*1000);			(* Delay OFF *)
			6:	Cmd_Buf_U16:=ADR(Cmd_Buf[8]);
				CIR06.OnDelay := DWORD_TO_TIME((Cmd_Buf_U16^)*60*1000);			(* Delay ON*)
				Cmd_Buf_U16:=ADR(Cmd_Buf[10]);
				CIR06.OffDelay := DWORD_TO_TIME((Cmd_Buf_U16^)*60*1000);			(* Delay OFF *)
			7:	Cmd_Buf_U16:=ADR(Cmd_Buf[8]);
				CIR07.OnDelay := DWORD_TO_TIME((Cmd_Buf_U16^)*60*1000);			(* Delay ON*)
				Cmd_Buf_U16:=ADR(Cmd_Buf[10]);
				CIR07.OffDelay := DWORD_TO_TIME((Cmd_Buf_U16^)*60*1000);			(* Delay OFF *)

		END_CASE


	5: (* GET Tempi delay On Off Circolatori *)
		Cmd_RLen:=4;
			CASE Cmd_ObjIdx OF


			1:	j:=DWORD_TO_WORD(TIME_TO_DWORD((CIR01.OnDelay)/60/1000));
				TxLen:=TxLen+RAWTOHEX(ADR(j),2,ADR(TxData[TxLen]));
				j:=DWORD_TO_WORD(TIME_TO_DWORD((CIR01.OffDelay)/60/1000));
				TxLen:=TxLen+RAWTOHEX(ADR(j),2,ADR(TxData[TxLen]));
			2: 	j:=DWORD_TO_WORD(TIME_TO_DWORD((CIR02.OnDelay)/60/1000));
				TxLen:=TxLen+RAWTOHEX(ADR(j),2,ADR(TxData[TxLen]));
				j:=DWORD_TO_WORD(TIME_TO_DWORD((CIR02.OffDelay)/60/1000));
				TxLen:=TxLen+RAWTOHEX(ADR(j),2,ADR(TxData[TxLen]));
			3:	j:=DWORD_TO_WORD(TIME_TO_DWORD((CIR03.OnDelay)/60/1000));
				TxLen:=TxLen+RAWTOHEX(ADR(j),2,ADR(TxData[TxLen]));
				j:=DWORD_TO_WORD(TIME_TO_DWORD((CIR03.OffDelay)/60/1000));
				TxLen:=TxLen+RAWTOHEX(ADR(j),2,ADR(TxData[TxLen]));
			4: 	j:=DWORD_TO_WORD(TIME_TO_DWORD((CIR04.OnDelay)/60/1000));
				TxLen:=TxLen+RAWTOHEX(ADR(j),2,ADR(TxData[TxLen]));
				j:=DWORD_TO_WORD(TIME_TO_DWORD((CIR04.OffDelay)/60/1000));
				TxLen:=TxLen+RAWTOHEX(ADR(j),2,ADR(TxData[TxLen]));
			5:	j:=DWORD_TO_WORD(TIME_TO_DWORD((CIR05.OnDelay)/60/1000));
				TxLen:=TxLen+RAWTOHEX(ADR(j),2,ADR(TxData[TxLen]));
				j:=DWORD_TO_WORD(TIME_TO_DWORD((CIR05.OffDelay)/60/1000));
				TxLen:=TxLen+RAWTOHEX(ADR(j),2,ADR(TxData[TxLen]));
			6: 	j:=DWORD_TO_WORD(TIME_TO_DWORD((CIR06.OnDelay)/60/1000));
				TxLen:=TxLen+RAWTOHEX(ADR(j),2,ADR(TxData[TxLen]));
				j:=DWORD_TO_WORD(TIME_TO_DWORD((CIR06.OffDelay)/60/1000));
				TxLen:=TxLen+RAWTOHEX(ADR(j),2,ADR(TxData[TxLen]));
			7: 	j:=DWORD_TO_WORD(TIME_TO_DWORD((CIR07.OnDelay)/60/1000));
				TxLen:=TxLen+RAWTOHEX(ADR(j),2,ADR(TxData[TxLen]));
				j:=DWORD_TO_WORD(TIME_TO_DWORD((CIR07.OffDelay)/60/1000));
				TxLen:=TxLen+RAWTOHEX(ADR(j),2,ADR(TxData[TxLen]));

		END_CASE






ELSE
	Cmd_R:=3;
END_CASE
END_ACTION
ACTION Cmd_CRON:
(* Check index *)
IF Cmd_ObjIdx<1 OR Cmd_ObjIdx>250 THEN
	Cmd_R:=2;
	RETURN;
END_IF

(* Process command *)
CASE Cmd_C OF


	1: (* GET PROFILE *)
		IF Cmd_CLen<>3 THEN
			Cmd_R:=4;
		ELSE
			(* Load profile *)
			CronEd.CN_Sel:=WORD_TO_BYTE(Cmd_ObjIdx);
			Cmd_Buf_U16:=ADR(Cmd_Buf[8]);
			CronEd.CN_YSel:=Cmd_Buf_U16^;
			IF Cmd_Buf[10]<=10 THEN
				CronEd.PR_Sel:=Cmd_Buf[10];
				CronEd.PR_Load_Exe();
				(* Response data *)
				Cmd_RLen:=192;
				TxLen:=TxLen+RAWTOHEX(ADR(CronEd.PR.Setpoint),192,ADR(TxData[TxLen]));
			ELSE
				Cmd_R:=6;
			END_IF
		END_IF

	2: (* SET PROFILE *)
		IF Cmd_CLen<>(3+192) THEN
			Cmd_R:=4;
		ELSE
			(* Save profile *)
			CronEd.CN_Sel:=WORD_TO_BYTE(Cmd_ObjIdx);
			Cmd_Buf_U16:=ADR(Cmd_Buf[8]);
			CronEd.CN_YSel:=Cmd_Buf_U16^;
			IF Cmd_Buf[10]<=10 THEN
				CronEd.PR_Sel:=Cmd_Buf[10];
				MEMCPY(ADR(Cmd_Buf[11]),ADR(CronEd.PR.Setpoint),192);
				CronEd.PR_Save_Exe();
			ELSE
				Cmd_R:=6;
			END_IF
		END_IF

	5: (* GET CALENDAR MONTH *)
		IF Cmd_CLen<>3 THEN
			Cmd_R:=4;
		ELSE
			(* Load calendar *)
			CronEd.CN_Sel:=WORD_TO_BYTE(Cmd_ObjIdx);
			Cmd_Buf_U16:=ADR(Cmd_Buf[8]);
			CronEd.CN_YSel:=Cmd_Buf_U16^;
			IF Cmd_Buf[10]>=1 AND Cmd_Buf[10]<=12 THEN
				CronEd.CA_Sel:=Cmd_Buf[10];
				CronEd.CA_Load_Exe();
				(* Response data *)
				Cmd_RLen:=32;
				TxLen:=TxLen+RAWTOHEX(ADR(CronEd.CA.Profile),32,ADR(TxData[TxLen]));
			ELSE
				Cmd_R:=6;
			END_IF
		END_IF

	6: (* SET CALENDAR MONTH *)
		IF Cmd_CLen<>(3+32) THEN
			Cmd_R:=4;
		ELSE
			(* Save calendar *)
			CronEd.CN_Sel:=WORD_TO_BYTE(Cmd_ObjIdx);
			Cmd_Buf_U16:=ADR(Cmd_Buf[8]);
			CronEd.CN_YSel:=Cmd_Buf_U16^;
			IF Cmd_Buf[10]>=1 AND Cmd_Buf[10]<=12 THEN
				CronEd.CA_Sel:=Cmd_Buf[10];
				MEMCPY(ADR(Cmd_Buf[11]),ADR(CronEd.CA.Profile),32);
				CronEd.CA_Save_Exe();
			ELSE
				Cmd_R:=6;
			END_IF
		END_IF

	9: (* CRON RESTART *)
		CASE Cmd_ObjIdx OF
			(*1: CRON01.InitOK:=FALSE;*)
			1: THER01.InitOK:=FALSE;
			2: THER02.InitOK:=FALSE;
			3: THER03.InitOK:=FALSE;
			4: THER04.InitOK:=FALSE;
			5: THER05.InitOK:=FALSE;
			250: THER250.InitOK:=FALSE;

		END_CASE

	10: (* SET Isteresi  *)
		CASE Cmd_ObjIdx OF
			1:	Cmd_Buf_U16:=ADR(Cmd_Buf[8]);
				THER01.Histeresys := Cmd_Buf_U16^; 			(* Isteresi*)
			2:	Cmd_Buf_U16:=ADR(Cmd_Buf[8]);
				THER02.Histeresys := Cmd_Buf_U16^; 			(* Isteresi*)
			3:	Cmd_Buf_U16:=ADR(Cmd_Buf[8]);
				THER03.Histeresys := Cmd_Buf_U16^; 			(* Isteresi*)
			4:	Cmd_Buf_U16:=ADR(Cmd_Buf[8]);
				THER04.Histeresys := Cmd_Buf_U16^; 			(* Isteresi*)
			5:	Cmd_Buf_U16:=ADR(Cmd_Buf[8]);
				THER05.Histeresys := Cmd_Buf_U16^; 			(* Isteresi*)
			250:	Cmd_Buf_U16:=ADR(Cmd_Buf[8]);
				THER250.Histeresys := Cmd_Buf_U16^; 			(* Isteresi*)
		END_CASE

	11: (* GET isteresi *)
		Cmd_RLen:=2;
		CASE Cmd_ObjIdx OF


			1: j:=(THER01.Histeresys);
				TxLen:=TxLen+RAWTOHEX(ADR(j),2,ADR(TxData[TxLen]));
			2: j:=(THER02.Histeresys);
				TxLen:=TxLen+RAWTOHEX(ADR(j),2,ADR(TxData[TxLen]));
			3: j:=(THER03.Histeresys);
				TxLen:=TxLen+RAWTOHEX(ADR(j),2,ADR(TxData[TxLen]));
			4: j:=(THER04.Histeresys);
				TxLen:=TxLen+RAWTOHEX(ADR(j),2,ADR(TxData[TxLen]));
			5: j:=(THER05.Histeresys);
				TxLen:=TxLen+RAWTOHEX(ADR(j),2,ADR(TxData[TxLen]));
			250: j:=(THER250.Histeresys);
				TxLen:=TxLen+RAWTOHEX(ADR(j),2,ADR(TxData[TxLen]));

		END_CASE
ELSE
	Cmd_R:=3;
END_CASE
END_ACTION
ACTION Cmd_CTL:
IF Cmd_ObjIdx<1 OR Cmd_ObjIdx>2 THEN
	Cmd_R:=2;
	RETURN;
END_IF

(* Process command *)
CASE Cmd_C OF


	0:	(* Comando limiti contalitri *)
		CASE Cmd_ObjIdx OF

		1: (* Scrittura Limite accettabile di pedite *)
			Cmd_Buf_U16:=ADR(Cmd_Buf[8]);
			CTL01.LimiteMaxPerdita:= Cmd_Buf_U16^;

		END_CASE

ELSE
	Cmd_R:=3;
END_CASE
END_ACTION
ACTION Cmd_SYS:
(* Check index *)
IF Cmd_ObjIdx<>0 THEN
	Cmd_R:=2;
	RETURN;
END_IF

(* Process command *)
CASE Cmd_C OF

	0: (* ECHO *)
		IF Cmd_CLen<>0 THEN
			TxLen:=0;
		END_IF

	1: (* LOG REQUEST *)
		LogTrig();

	2: (* REARM *)
		Sys.Warning:=FALSE;
		Sys.Alarm:=FALSE;
		Sys.AlarmStop:=FALSE;

	3: (* GET INFO1 *)
		Cmd_RLen:=6;
		TxLen:=TxLen+RAWTOHEX(ADR(Plant_SN),4,ADR(TxData[TxLen]));
		TxLen:=TxLen+RAWTOHEX(ADR(Plant_SW_VER),2,ADR(TxData[TxLen]));


	4: (*  Scrivo i Parametri gestione Impianto   *)

			Cmd_Buf_U16:=ADR(Cmd_Buf[8]);
			DelayAllarmeTemperaturaNonRaggiunta := Cmd_Buf_U16^; 			(* Ritardo Allarme dall'avvio Caldaia*)
			Cmd_Buf_U16:=ADR(Cmd_Buf[10]);
			DeltaInterventoAllarmeTempeaturaNonRaggiuta := Cmd_Buf_U16^;	(* Delta Soglia Temperatura per Allarme Temperatura Non Raggiunta *)
			Cmd_Buf_U16:=ADR(Cmd_Buf[12]);
			OffsetSetPointManuale := Cmd_Buf_U16^; 							(* Offest Perdite Scambiatore 1  *)
			Cmd_Buf_U16:=ADR(Cmd_Buf[14]);
			OffsetSetPointManuale2 := Cmd_Buf_U16^; 						(* Offest Perdite Scambiatore 1  *)
			Cmd_Buf_U16:=ADR(Cmd_Buf[12]);
			BitAbilitaBoost :=INT_TO_BOOL( Cmd_Buf_U16^); 					(* Abilitazione controllo Boost  *)
			Cmd_Buf_U16:=ADR(Cmd_Buf[14]);
			RifOffsetBoost := Cmd_Buf_U16^; 								(* Offset al Setpoint della Caldaia per azione di Boost  *)


	5: (*  Leggi i parametri gestione Impianto  *)

			Cmd_RLen:=18;
			j:=(DelayAllarmeTemperaturaNonRaggiunta);   				(* Ritardo Allarme dall'avvio Caldaia*)
			TxLen:=TxLen+RAWTOHEX(ADR(j),2,ADR(TxData[TxLen]));
			j:=(DeltaInterventoAllarmeTempeaturaNonRaggiuta);			(* Delta Soglia Temperatura per Allarme Temperatura Non Raggiunta *)
			TxLen:=TxLen+RAWTOHEX(ADR(j),2,ADR(TxData[TxLen]));
			j:=(OffsetSetPointManuale);									(* Offest Perdite Scambiatore 1  *)
			TxLen:=TxLen+RAWTOHEX(ADR(j),2,ADR(TxData[TxLen]));
			j:=(OffsetSetPointManuale2);								(* Offest Perdite Scambiatore 2  *)
			TxLen:=TxLen+RAWTOHEX(ADR(j),2,ADR(TxData[TxLen]));
			j:=BOOL_TO_INT(BitAbilitaBoost);							(* Abilitazione controllo Boost  *)
			TxLen:=TxLen+RAWTOHEX(ADR(j),2,ADR(TxData[TxLen]));
			j:=BOOL_TO_INT(BitAbilitaBoost);										(* Offset al Setpoint della Caldaia per azione di Boost   *)
			TxLen:=TxLen+RAWTOHEX(ADR(j),2,ADR(TxData[TxLen]));




	6: (*  Scrivo i Parametri gestione Impianto - Antigelo   *)

			Cmd_Buf_U16:=ADR(Cmd_Buf[8]);
			SogliaMinStartAntigelo := Cmd_Buf_U16^; 			(* Soglia mininma Start Antigelo *)
			Cmd_Buf_U16:=ADR(Cmd_Buf[10]);
			SogliaMinStopAntigelo := Cmd_Buf_U16^;				(* Soglia Massima Stop Antigelo *)
			Cmd_Buf_U16:=ADR(Cmd_Buf[12]);
			BitAbilitaAntigelo :=INT_TO_BOOL( Cmd_Buf_U16^); 	(* Abilitazione Antigelo  *)

	7: (*  Leggi i parametri gestione Impianto - Antigelo *)

			Cmd_RLen:=14;
			j:=(SogliaMinStartAntigelo); 							(* Soglia mininma Start Antigelo *)
			TxLen:=TxLen+RAWTOHEX(ADR(j),2,ADR(TxData[TxLen]));
			j:=(SogliaMinStopAntigelo);								(* Soglia Massima Stop Antigelo *)
			TxLen:=TxLen+RAWTOHEX(ADR(j),2,ADR(TxData[TxLen]));
			j:=BOOL_TO_INT(BitAbilitaAntigelo);						(* Abilitazione Antigelo  *)
			TxLen:=TxLen+RAWTOHEX(ADR(j),2,ADR(TxData[TxLen]));

(*	10: (*  Scrivo i Parametri per la gestione della velocità dei circolatori sui primari   *)

			Cmd_Buf_U16:=ADR(Cmd_Buf[8]);
			PercVelMin := Cmd_Buf_U16^;
			Cmd_Buf_U16:=ADR(Cmd_Buf[10]);
			PercVelMax := Cmd_Buf_U16^;
			Cmd_Buf_U16:=ADR(Cmd_Buf[12]);
			ErroreTempMax := Cmd_Buf_U16^;
			Cmd_Buf_U16:=ADR(Cmd_Buf[14]);
			ErroreTempMin := Cmd_Buf_U16^;

	11: (*  Leggo i Parametri per la gestione della velocità dei circolatori sui primari   *)

			Cmd_RLen:=8;
			j:=(PercVelMin);
			TxLen:=TxLen+RAWTOHEX(ADR(j),2,ADR(TxData[TxLen]));
			j:=(PercVelMax);
			TxLen:=TxLen+RAWTOHEX(ADR(j),2,ADR(TxData[TxLen]));
			j:=(ErroreTempMax);
			TxLen:=TxLen+RAWTOHEX(ADR(j),2,ADR(TxData[TxLen]));
			j:=(ErroreTempMin);
			TxLen:=TxLen+RAWTOHEX(ADR(j),2,ADR(TxData[TxLen]));


	12: (*  Scrivo i Parametri per la gestione della velocità dei circolatori sui primari   *)


				Cmd_Buf_U16:=ADR(Cmd_Buf[8]);
				CAS01.DeltaTempThr := Cmd_Buf_U16^;
				Cmd_Buf_U16:=ADR(Cmd_Buf[10]);
				CAS01.Tmonitor_Off := DWORD_TO_TIME((Cmd_Buf_U16^)*60*1000);
				Cmd_Buf_U16:=ADR(Cmd_Buf[12]);
				CAS01.Tmonitor_On := DWORD_TO_TIME((Cmd_Buf_U16^)*60*1000);

	13: (*  Leggo i Parametri per la gestione della velocità dei circolatori sui primari   *)


				Cmd_RLen:=6;
				j:=(CAS01.DeltaTempThr);
				TxLen:=TxLen+RAWTOHEX(ADR(j),2,ADR(TxData[TxLen]));
				j:=DWORD_TO_WORD(TIME_TO_DWORD((CAS01.Tmonitor_Off)/60/1000));
				TxLen:=TxLen+RAWTOHEX(ADR(j),2,ADR(TxData[TxLen]));
				j:=DWORD_TO_WORD(TIME_TO_DWORD((CAS01.Tmonitor_On)/60/1000));
				TxLen:=TxLen+RAWTOHEX(ADR(j),2,ADR(TxData[TxLen]));


*)


	14: (*  Imposto data e ora del PLC  *)


			Cmd_Buf_U16:=ADR(Cmd_Buf[8]);
			SetAnno:= Cmd_Buf_U16^; 												(* Anno *)
			Cmd_Buf_U16:=ADR(Cmd_Buf[10]);
			SetMese:= Cmd_Buf_U16^;												 	(* mese *)
			Cmd_Buf_U16:=ADR(Cmd_Buf[12]);
			SetGiorno:=( Cmd_Buf_U16^);											 	(* Giorno *)
			Cmd_Buf_U16:=ADR(Cmd_Buf[14]);
			SetOra:=( Cmd_Buf_U16^); 												(* ora *)
			Cmd_Buf_U16:=ADR(Cmd_Buf[16]);
			SetMinuti:= ( Cmd_Buf_U16^);										 	(* Minuti *)
			Cmd_Buf_U16:=ADR(Cmd_Buf[18]);
			SetSecondi:= ( Cmd_Buf_U16^);										 	(* secondi *)

	(*		SysRtcSetTime(SetDataTime(DWORD_TO_INT(ADR(Cmd_Buf[8])),				(* Anno *)
										DWORD_TO_INT(ADR(Cmd_Buf[10])),				(* mese *)
										DWORD_TO_INT(ADR(Cmd_Buf[11])),				(* Giorno *)
										DWORD_TO_INT(ADR(Cmd_Buf[12])),				(* ora *)
										DWORD_TO_INT(ADR(Cmd_Buf[13])),				(* Minuti *)
										DWORD_TO_INT(ADR(Cmd_Buf[14]))				(* secondi *)
										)); *)

		SysRtcSetTime((SetDataTime(SetAnno,SetMese,SetGiorno,SetOra,SetMinuti,SetSecondi)));


ELSE
	Cmd_R:=3;
END_CASE
END_ACTION
ACTION Cmd_VRD:
(* Check index *)
IF Cmd_ObjIdx<1 OR Cmd_ObjIdx>2 THEN
	Cmd_R:=2;
	RETURN;
END_IF

(* Process command *)
CASE Cmd_C OF

	1: (* GET CLIMATIC *)
		Cmd_RLen:=20;
		FOR i:=0 TO 4 DO
			IF Cmd_ObjIdx=1 THEN
				j:=DINT_TO_INT(VRD01_Clima.Points[i].X);
			ELSE
				j:=DINT_TO_INT(VRD02_Clima.Points[i].X);
			END_IF
			TxLen:=TxLen+RAWTOHEX(ADR(j),2,ADR(TxData[TxLen]));
			IF Cmd_ObjIdx=1 THEN
				j:=DINT_TO_INT(VRD01_Clima.Points[i].Y);
			ELSE
				j:=DINT_TO_INT(VRD02_Clima.Points[i].Y);
			END_IF
			TxLen:=TxLen+RAWTOHEX(ADR(j),2,ADR(TxData[TxLen]));
		END_FOR

	2: (* SET CLIMATIC *)
		IF Cmd_CLen<>20 THEN
			Cmd_R:=4;
		ELSE
			FOR i:=0 TO 4 DO
				Cmd_Buf_INT:=ADR(Cmd_Buf[8+4*i]); j:=Cmd_Buf_INT^;
				IF Cmd_ObjIdx=1 THEN
					VRD01_Clima.Points[i].X:=INT_TO_DINT(j);
				ELSE
					VRD02_Clima.Points[i].X:=INT_TO_DINT(j);
				END_IF
				Cmd_Buf_INT:=ADR(Cmd_Buf[10+4*i]); j:=Cmd_Buf_INT^;
				IF Cmd_ObjIdx=1 THEN
					VRD01_Clima.Points[i].Y:=INT_TO_DINT(j);
				ELSE
					VRD02_Clima.Points[i].Y:=INT_TO_DINT(j);
				END_IF
			END_FOR
		END_IF

ELSE
	Cmd_R:=3;
END_CASE
END_ACTION
ACTION Command:
(* Default response OK/NODATA *)
Cmd_R:=0;
Cmd_RLen:=0;
TxLen:=16;

(* Check object *)
CASE Cmd_Obj OF

	EO_SYS:
		Cmd_SYS();

	EO_CAL:
		Cmd_CAL();

	EO_VRD:
		Cmd_VRD();

	EO_CRON:
		Cmd_CRON();

	EO_CIR:
		Cmd_CIR();

	EO_CTL:
		Cmd_CTL();


ELSE
	Cmd_R:=1;
END_CASE

(* Generate response *)
IF TxLen>0 THEN
	RAWTOHEX(ADR(Cmd_Obj)	,2,ADR(TxData[ 0]));
	RAWTOHEX(ADR(Cmd_ObjIdx),2,ADR(TxData[ 4]));
	RAWTOHEX(ADR(Cmd_R)		,2,ADR(TxData[ 8]));
	RAWTOHEX(ADR(Cmd_RLen)	,2,ADR(TxData[12]));
	TxTrig:=TRUE;
END_IF
END_ACTION

(* POU Utils Functions/TCPSERVER, ST *)
FUNCTION_BLOCK TCPSERVER
(***********************************************************************************************************	*)
(* Version: 1.6                                    			          											*)
(* Date: 11.02.2011                                   					          							    *)
(***********************************************************************************************************	*)
(* WAGO Kontakttechnik GmbH Hansastr. 27 32423 Minden(Westf.)													*)
(* Tel. +0049 571/887-0 Fax. +0049 571/887-0																	*)
(* Author: VB																									*)
(***********************************************************************************************************	*)
(*Description:	A TCP server to read and write data													       		*)
(*Historie:																										*)
(*Version 1.6: 11.02.2011: Changes according to 750-880/881											 			*)
(*Version 1.5: 27.11.2008 Bugfix allow reuse port																*)
(*Version 1.4: 13.10.2008 Bugfix transmitting large data														*)
(*Version 1.3: 15.01.2007 Changes according to FW11																*)
(*Version 1.2: 09.03.2006 Changes for socket handle 0											       			*)
(*Version 1.1: 14.02.2005 Release																				*)
(***********************************************************************************************************	*)
VAR CONSTANT
	STATE_INIT     				 : BYTE:= 0;
	STATE_OPEN     				 : BYTE:= 1;
	STATE_TX       				 : BYTE:= 20;
	STATE_RX       				 : BYTE:= 30;
	STATE_CLOSE    				 : BYTE:= 40;
	STATE_ERROR_TRAP		 	 : BYTE:= 200;
END_VAR
VAR_INPUT
	xEnable    					: BOOL;	 (* Set TRUE to enable function block *)
	wPortNumber					: WORD;  (* Port *)
	tServerTimeOut				: TIME:=t#50s;
	ptSendData					: POINTER TO ARRAY[0..MAX_SEND_TCP_SERVER] OF BYTE;
	diSendCount					: DINT;
END_VAR
VAR_OUTPUT
	xClientConnected  			: BOOL:= FALSE;
	diError 					: DINT:= 0;
END_VAR
(* Status Codes -----------------------------------------
	16#8001 => No socket descriptor available 
	16#8002 => SysSockBind fails 
	16#8003 => SysSockListen fails 
	16#8004 => switching to none blocking mode fails
	16#8005 => SysSockClose() returns FALSE 
    16#8006 => SysSockConnect() fails
    16#8007 => SysSockSend() fails
	16#8008 => error state machine 
	16#8009 => timeout while waiting for data from server 
	16#0001 => server waiting for client to establish connection
------------------------------------------------------------*)
VAR_IN_OUT
	xStartSend					: BOOL;
	aReceiveBuffer				: ARRAY [0..MAX_RECEIVE_TCP_SERVER] OF BYTE;
	diReceiveCount				: DINT;
END_VAR

VAR
	m_State    					: BYTE:= 0;
	m_ReceiveBuffer				: ARRAY [0..MAX_RECEIVE_TCP_SERVER_SOCKET] OF BYTE;
	m_ServerSocket				: DINT:= SOCKET_INVALID;
	m_Socket					: DINT:= SOCKET_INVALID;
	m_AddressInfo				: SOCKADDRESS;
	m_BytesReceived				: DINT;
	m_diReturn					: DINT;
	m_xReturn					: BOOL;
	m_SizeSockadr				: DWORD;
	m_ConnectionWatchdog		: TON;
	m_Flags						: DINT;
	m_NoneBlocking   			: DINT:= 1;
	m_Blocking   				: DINT:= 0;
	i							: INT;
	m_count						: DINT;
	diOption					: DINT := 1;
	on: DINT;
END_VAR
IF xEnable THEN
	CASE m_State OF
		STATE_INIT:
			(* Create Socket *)
			m_ServerSocket:= SysSockCreate( SOCKET_AF_INET, SOCKET_STREAM, 0);
			IF m_ServerSocket = SOCKET_INVALID THEN
				(* *)
				diError:= 16#8001;
				m_State:= STATE_ERROR_TRAP;
				RETURN;
			ELSE
				;
			END_IF
			(* Address bindings *)
			(********************)
			on:=1;
			SysSockSetOption( m_ServerSocket, SOCKET_SOL, SOCKET_SO_REUSEADDR, ADR(on), SIZEOF(on) );

			m_AddressInfo.sin_family:= SOCKET_AF_INET;
			m_AddressInfo.sin_port  := SysSockHtons( wPortNumber);
			m_AddressInfo.sin_addr  := SOCKET_INADDR_ANY;
			IF NOT SysSockBind( m_ServerSocket, ADR(m_AddressInfo), SIZEOF(m_AddressInfo)) THEN
				diError:= 16#8002;
				m_State:= STATE_ERROR_TRAP;
				RETURN;
			END_IF
			(* Wait for connections *)
			(************************)
			IF NOT SysSockListen( m_ServerSocket, 1) THEN
				diError:= 16#8003;
				m_State:= STATE_ERROR_TRAP;
			END_IF

			(* Puts SOCKET in NonBlocking mode *)
			m_diReturn:= SysSockIoctl( m_ServerSocket, SOCKET_FIONBIO, ADR(m_NoneBlocking));

			m_State:= STATE_OPEN;


		STATE_OPEN: 	(* Waiting for incomming connection *)
				m_SizeSockadr:=SIZEOF(m_AddressInfo);
				m_Socket:= SysSockAccept( m_ServerSocket, ADR(m_AddressInfo), ADR(m_SizeSockadr));
				diError:=State_open;
				IF m_Socket <> SOCKET_INVALID THEN
					xClientConnected:=TRUE;
					(*Set Push-Bit:new V1.5*)
					IF ADR(%MW0)=16#30000000  OR ADR(%MW0)=16#20000000 THEN (*841 or 881*)
						SysSockSetOption(
							diSocket:=m_Socket,
							diLevel:=6,
							diOption:=SOCKET_TCP_NODELAY,
							pOptionValue:=ADR(diOption),
							diOptionLength:=SIZEOF(diOption));
					ELSE
							;
					END_IF
					SysSockIoctl( m_Socket, SOCKET_FIONBIO, ADR(m_NoneBlocking));
					m_State:= STATE_RX;
					diError:=0;
				END_IF

		STATE_RX:
					m_BytesReceived:= SysSockRecv( m_Socket, ADR(m_ReceiveBuffer), SIZEOF(m_ReceiveBuffer), 0);
					CASE m_BytesReceived OF
					-1:(*no data available or error occured*)
						m_ConnectionWatchdog(IN:=TRUE , PT:=tServerTimeOut );
						IF m_connectionWatchdog.Q THEN
							m_State:= STATE_CLOSE;
							m_ConnectionWatchdog(IN:=FALSE);(*reset connection watchdog*)
							diError := 16#8009;
						END_IF
					0:(* socket was "gracefully closed"  *)
						m_State:= STATE_CLOSE;
						diError := 16#8003;
					ELSE
						(* Copy received data into receive buffer *)
						(********************************)
						FOR i:= 0 TO DINT_TO_INT(m_BytesReceived	)-1 DO
							aReceiveBuffer[diReceiveCount]:= m_ReceiveBuffer[i];
							diReceiveCount:=(diReceiveCount+1) MOD SIZEOF(aReceiveBuffer);
						END_FOR

						m_ConnectionWatchdog(IN:=FALSE);(*reset connection watchdog*)
					END_CASE

				(*send data*)
				IF xStartSend	 THEN
					m_State := STATE_TX;
				END_IF

	STATE_TX:	 (* send TCP-message *)
		m_diReturn := SysSockSend(diSocket := m_Socket,
								  pbyBuffer := ADR(ptSendData^[m_count]),(*geändert V1.4 bisher: [0] *)
								  diBufferSize := diSendCount-m_count,
								  diFlags :=m_Flags);
		CASE m_diReturn OF
		-1:	(* ERROR or data could not yet be send (V1.3 due to new FW11) *)
			m_ConnectionWatchdog(IN:=TRUE , PT:=tServerTimeOut );
			IF m_connectionWatchdog.Q THEN
				m_State:= STATE_CLOSE;
				m_ConnectionWatchdog(IN:=FALSE);(*reset connection watchdog*)
				diError := 16#8007;
			END_IF
		0: (* socket was "gracefully closed"  *)
			m_State := STATE_CLOSE;
			diError := 16#8003;
		ELSE (* succesful *)
			m_count:=m_count+m_diReturn;
			IF m_count>=diSendCount THEN
				diError := 16#0000;
				m_State := STATE_RX;
				m_count:=0;
				xStartSend:=FALSE;
			END_IF
			m_ConnectionWatchdog(IN:=FALSE);(*reset connection watchdog*)
		END_CASE


		STATE_CLOSE:	(* Close the server *)

		IF ADR(%MW0)=16#30000000  OR ADR(%MW0)=16#20000000 THEN (*841 or 881*)
			;
		ELSE
			IF m_Socket>=0 THEN
				SysSockShutdown(m_Socket, 0);;(*870*)
			END_IF
		END_IF
		IF m_Socket>=0 THEN
			SysSockClose( m_Socket);
		END_IF
		xClientConnected:= FALSE;
		m_State:= STATE_OPEN; (* Try to open the server again *)
		m_ConnectionWatchdog(IN:=FALSE);(*reset connection watchdog*)

		STATE_ERROR_TRAP: (* Error Read/Write socket  *)
			m_State:= STATE_ERROR_TRAP;

	ELSE  (* Bad FSM code trap  *)
			m_State:= STATE_ERROR_TRAP;
			diError:= 16#8008;
	END_CASE;
ELSE
	IF m_State <> STATE_INIT THEN
		IF ADR(%MW0)=16#30000000  OR ADR(%MW0)=16#20000000 THEN (*841 or 881*)
			;
		ELSE
			IF m_Socket>=0 THEN
				SysSockShutdown(m_Socket, 0);;(*870*)
			END_IF
		END_IF
		IF m_Socket>=0 THEN
			SysSockClose( m_Socket);
		END_IF
		IF ADR(%MW0)=16#30000000  OR ADR(%MW0)=16#20000000 THEN (*841 or 881*)
			;
		ELSE
			IF m_ServerSocket>=0 THEN
				SysSockShutdown(m_ServerSocket, 0);;(*870*)
			END_IF
		END_IF
		IF m_ServerSocket>=0 THEN
			SysSockClose( m_ServerSocket);
		END_IF
		xClientConnected:= FALSE;
		diError:= 0;
		m_State:= STATE_init; (* Try to open the server again *)
		m_ConnectionWatchdog(IN:=FALSE);(*reset connection watchdog*)
	END_IF
END_IF
END_FUNCTION_BLOCK

(* POU TCP_Logger/LogEv, ST *)
FUNCTION LogEv : BOOL
VAR_INPUT
	Level	: en_Logger_ErrLev;
	Object  : en_SYS_Objects;
	Index	: WORD;
	Error	: WORD;
	Message : STRING;
END_VAR
VAR
	s1 : STRING(160);
	i  : INT;
END_VAR
(* Execute error level operations *)

Sys.Alarm:=Lamp.SistemaInAllarme;
Sys.Warning:=Lamp.SistemaWarning;


(* Fill lastlog list *)
s1:=CONCAT(Sys.Time_LogString,';Lev=');
s1:=CONCAT(s1,INT_TO_STRING(Level));
s1:=CONCAT(s1,';Obj=');
s1:=CONCAT(s1,INT_TO_STRING(Object));
s1:=CONCAT(s1,';Idx=');
s1:=CONCAT(s1,WORD_TO_STRING(Index));
s1:=CONCAT(s1,';Err=');
s1:=CONCAT(s1,WORD_TO_STRING(Error));
Sys.LastLogs_Dat[Sys.LastLogs_Idx]:=s1;
Sys.LastLogs_Msg[Sys.LastLogs_Idx]:=Message;
Sys.LastLogs_Idx:=Sys.LastLogs_Idx+1;
IF Sys.LastLogs_Idx>5 THEN Sys.LastLogs_Idx:=0; END_IF

(*---------------------------------------------------------------*)
	Logger_Head();
(*---------------------------------------------------------------*)

(* Insert ERR *)
s1:=CONCAT('&ERR=',INT_TO_STRING(Level));
s1:=CONCAT(s1,';');
s1:=CONCAT(s1,INT_TO_STRING(Object));
s1:=CONCAT(s1,';');
s1:=CONCAT(s1,WORD_TO_STRING(Index));
s1:=CONCAT(s1,';');
s1:=CONCAT(s1,WORD_TO_STRING(Error));
s1:=CONCAT(s1,';');
ADDSTRING(ADR(Logger.TData), ADR(s1), Logger.TLen);
s1:=Message;
STR_NOSPACES(ADR(s1));
ADDSTRING(ADR(Logger.TData), ADR(s1), Logger.TLen);

(*---------------------------------------------------------------*)
	Logger_Send();
(*---------------------------------------------------------------*)
END_FUNCTION

(* POU TCP_Logger/Logger_Head, ST *)
FUNCTION Logger_Head : BOOL
VAR
	s1 : STRING(160);
	i  : BYTE;
END_VAR
Logger.TLen:=0;
(* Set GET header *)
ADDSTRING(ADR(Logger.TData), ADR(Logger_GETSTART), Logger.TLen);

(* Insert Header *)
s1:=INSERT('ID=&V=1&D=',DWORD_TO_STRING(Plant_SN),3);
s1:=CONCAT(s1,REPLACE(Sys.Time_LogString,'T',1,11));
(*s1:=CONCAT(s1,Sys.Time_LogString) *)
s1:=CONCAT(s1,'&S=');
IF Sys.Alarm THEN i:=2; ELSIF Sys.Warning THEN i:=1; ELSE i:=0; END_IF
s1:=CONCAT(s1,BYTE_TO_STRING(i));
ADDSTRING(ADR(Logger.TData), ADR(s1), Logger.TLen);
END_FUNCTION

(* POU Utils Functions/ADDSTRING, ST *)
FUNCTION ADDSTRING : BOOL
VAR_INPUT
	pTxData: POINTER TO BYTE;
	pString: POINTER TO BYTE;
END_VAR
VAR_IN_OUT
	TxLen: DINT;
END_VAR
VAR
END_VAR
pTxData:=pTxData+TxLen;
WHILE pString^<>0 DO
	pTxData^:=pString^;
	pString:=pString+1;
	pTxData:=pTxData+1;
	TxLen:=TxLen+1;
END_WHILE
END_FUNCTION

(* POU Utils Functions/STR_NOSPACES, ST *)
FUNCTION STR_NOSPACES : BOOL (* Replace spaces and bad chars with allowed ones, used as HTTP-GET validator *)
VAR_INPUT
	pString: POINTER TO BYTE;
END_VAR
VAR
END_VAR
WHILE pString^<>0 DO
	IF pString^=16#20 (* space *) THEN pString^:=16#5F; (*'_'*) END_IF
	pString:=pString+1;
END_WHILE
END_FUNCTION

(* POU TCP_Logger/Logger_Send, ST *)
FUNCTION Logger_Send : BOOL
VAR
	hFile: 	DWORD;
	pos:	DWORD;
END_VAR
(* Finalize string *)
ADDSTRING(ADR(Logger.TData), ADR(Logger_GETEND), Logger.TLen);

(* Read log position *)
pos:=SysFileGetSize(Logger_DataFile);
(* Check log size, bckup and erase if no pending messages *)
IF pos>5000000(*5M*) THEN
	hFile:=SysFileOpen(Logger_IndexFile,'r');
	IF hFile=0 THEN
		SysFileDelete(Logger_DataFileOld);
		SysFileRename(Logger_DataFile,Logger_DataFileOld);
		pos:=0;
	ELSE
		SysFileClose(hFile);
	END_IF
END_IF
(* Write message on log file *)
hFile:=SysFileOpen(Logger_DataFile,'a');
IF hFile<>0 THEN
	SysFileWrite(hFile, ADR(Logger.TData), Logger.TLen);
	SysFileClose(hFile);
ELSE
	Sys.Warning:=TRUE;
END_IF


(* Check logger status *)
IF Logger.SendReq=FALSE THEN
	(* Set log position for recovery *)
	Logger.SendIdx:=pos;
	(* Copy message data *)
	MEMCPY(ADR(Logger.TData),ADR(Logger.SendData),DINT_TO_WORD(Logger.TLen));
	Logger.SendLen:=Logger.TLen;
	(* Trigger request *)
	Logger.SendReq:=TRUE;
ELSE
	(* Add message position+size in recovery indexes *)
	hFile:=SysFileOpen(Logger_IndexFile,'a');
	SysFileWrite(hFile, ADR(pos), SIZEOF(pos));
	SysFileWrite(hFile, ADR(Logger.TLen), SIZEOF(Logger.TLen));
	SysFileClose(hFile);
END_IF
END_FUNCTION

(* POU Utils Functions/MEMCPY, ST *)
FUNCTION MEMCPY:BOOL
VAR_INPUT
	pSourceAddress:POINTER TO ARRAY[1..2] OF BYTE;
	pDestinationAddress:POINTER TO ARRAY[1..2] OF BYTE;
	BytesToCopy:WORD;
END_VAR
VAR
END_VAR
WHILE (BytesToCopy > 0) DO
	pDestinationAddress^[1]:=pSourceAddress^[1]; (* copy bytes from source to destination *)
	pDestinationAddress:=ADR(pDestinationAddress^[2]); (* increment destination *)
	pSourceAddress:=ADR(pSourceAddress^[2]);(* increment source *)
	BytesToCopy:=BytesToCopy -1; (* decrement number of bytes to copy *)
END_WHILE
END_FUNCTION

(* POU Utils Functions/HEXTORAW, ST *)
FUNCTION HEXTORAW : WORD
VAR_INPUT
	pString		: POINTER TO BYTE;
	StringLen	: WORD;
	pData		: POINTER TO BYTE;
END_VAR
VAR
	xl: WORD;
	xi: WORD;
	xr: BYTE;
END_VAR
xl:=0;
xi:=0;

WHILE xi<StringLen DO

	IF pString^>=97 AND pString^<=102 THEN
		xr := pString^ - 87;
	ELSIF pString^>=65 AND pString^<=70 THEN
		xr := pString^ - 55;
	ELSIF pString^>=48 AND pString^<=57 THEN
		xr := pString^ - 48;
	ELSE
		xr := 16;
	END_IF

	IF xr<16 THEN
		IF (xi AND 1)=0 THEN
			pData^ := xr * 16;
		ELSE
			pData^ := pData^ + xr;
			pData := pData + 1;
			xl := xl + 1;
		END_IF
	END_IF

	xi := xi + 1;
	pString := pString + 1;

END_WHILE

HEXTORAW:=xl;
END_FUNCTION

(* POU Utils Functions/RAWTOHEX, ST *)
FUNCTION RAWTOHEX : WORD
VAR_INPUT
	pData: POINTER TO BYTE;
	DataLen: WORD;
	pString: POINTER TO BYTE;
END_VAR
VAR
	xl: WORD;
END_VAR
xl:=0;

WHILE DataLen>0 DO

	pString^ := (pData^ / 16#10) + 48 + (((pData^ / 16#10)/10)*7);
	pString:=pString+1;
	pString^ := (pData^ AND 16#0F)  + 48 + (((pData^ AND 16#0F)/10)*7);
	pString:=pString+1;
	pData:=pData+1;
	DataLen:=DataLen-1;
	xl:=xl+2;

END_WHILE

(*pString^:=0;*)

RAWTOHEX:=xl;
END_FUNCTION

(* POU Utils Functions/GestioneDataTime_DaOscat/SetDataTime, ST *)
FUNCTION SetDataTime : DT
VAR_INPUT
	year : INT;
	month : INT;
	day : INT;
	hour : INT;
	minute : INT;
	second : INT;
END_VAR

VAR
	count : INT;
END_VAR
(* Creazione variabiletipo DT per creare Orario da dare al PLC *)


IF month > 2 THEN
	count := (month - 1) * 30;
	IF month > 7 THEN count := count + SHR(month - 3,1); ELSE count := count + SHR(month - 4,1); END_IF;
	(* chech for leap year and add one day if true *)
	IF SHL(year,14) = 0 THEN count := count + 1; END_IF;
ELSE
	count := (month - 1) * 31;
END_IF;


SetDataTime := DWORD_TO_DT(DATE_TO_DWORD( DWORD_TO_DATE((INT_TO_DWORD(count + day - 1) + SHR(INT_TO_DWORD(year) * 1461 - 2878169, 2)) * 86400))
				+ INT_TO_DWORD(SECOND)
				+ INT_TO_DWORD(MINUTE) * 60
				+ INT_TO_DWORD(HOUR) * 3600);
END_FUNCTION

(* POU Utils/USRLED_Update, ST *)
PROGRAM USRLED_Update
VAR
	OldStatus: en_SYS_Status;

	aFS : ARRAY [0..24] OF FLASHING_SEQUENCE :=
		(Colour:=GREEN,  Frequency:=1,   Relation:=128, Duration:=t#0s,    NextIndex:=0),  (* 0 => RUNNING *)
		(Colour:=ORANGE, Frequency:=1,   Relation:=128, Duration:=t#0s,    NextIndex:=1),  (* 1 => INIT *)
		(Colour:=RED,    Frequency:=4,   Relation:=128, Duration:=t#0s,    NextIndex:=2),  (* 2 => ERROR *)
		(Colour:=RED,    Frequency:=10,  Relation:=128, Duration:=t#0s,    NextIndex:=3),  (* 3 => ALARM *)
		(Colour:=ORANGE, Frequency:=200, Relation:=16,  Duration:=t#100ms, NextIndex:=11), (* 10 *)
		(Colour:=ORANGE, Frequency:=200, Relation:=32,  Duration:=t#100ms, NextIndex:=12),
		(Colour:=ORANGE, Frequency:=200, Relation:=64,  Duration:=t#100ms, NextIndex:=13),
		(Colour:=ORANGE, Frequency:=200, Relation:=128, Duration:=t#100ms, NextIndex:=14),
		(Colour:=ORANGE, Frequency:=200, Relation:=192, Duration:=t#100ms, NextIndex:=15),
		(Colour:=ORANGE, Frequency:=200, Relation:=128, Duration:=t#100ms, NextIndex:=16),
		(Colour:=ORANGE, Frequency:=200, Relation:=64,  Duration:=t#100ms, NextIndex:=17),
		(Colour:=ORANGE, Frequency:=200, Relation:=32,  Duration:=t#100ms, NextIndex:=18),
		(Colour:=ORANGE, Frequency:=200, Relation:=16,  Duration:=t#100ms, NextIndex:=19),
		(Colour:=ORANGE, Frequency:=200, Relation:=8,   Duration:=t#100ms, NextIndex:=10),
		(Colour:=GREEN,  Frequency:=200, Relation:=16,  Duration:=t#100ms, NextIndex:=21), (* 20 *)
		(Colour:=GREEN,  Frequency:=200, Relation:=32,  Duration:=t#100ms, NextIndex:=22),
		(Colour:=GREEN,  Frequency:=200, Relation:=64,  Duration:=t#100ms, NextIndex:=23),
		(Colour:=GREEN,  Frequency:=200, Relation:=128, Duration:=t#100ms, NextIndex:=24),
		(Colour:=GREEN,  Frequency:=200, Relation:=192, Duration:=t#100ms, NextIndex:=25),
		(Colour:=GREEN,  Frequency:=200, Relation:=128, Duration:=t#100ms, NextIndex:=26),
		(Colour:=GREEN,  Frequency:=200, Relation:=64,  Duration:=t#100ms, NextIndex:=27),
		(Colour:=GREEN,  Frequency:=200, Relation:=32,  Duration:=t#100ms, NextIndex:=28),
		(Colour:=GREEN,  Frequency:=200, Relation:=16,  Duration:=t#100ms, NextIndex:=29),
		(Colour:=GREEN,  Frequency:=200, Relation:=8,   Duration:=t#100ms, NextIndex:=20);

	pFS : POINTER TO FLASHING_SEQUENCE;


END_VAR
IF Sys.Status <> OldStatus THEN

	OldStatus:=Sys.Status;

	CASE OldStatus OF

		S_STARTUP:
			pFS:=ADR(aFS);
			SET_FLASHING_SEQUENCE(EN:=TRUE, POINTER_TO_POINTER_TO_ARRAY:=ADR(pFS));
			SET_FLASHING_SEQUENCE_INDEX(EN:=TRUE, IMMEDIATE:=FALSE, INDEX:=1);
			START_FLASHING_SEQUENCE(EN:=TRUE);

		S_RUNNING:
			SET_FLASHING_SEQUENCE_INDEX(EN:=TRUE, IMMEDIATE:=TRUE, INDEX:=0);

	END_CASE

END_IF
END_PROGRAM

(* POU Utils Functions/LINEAR_BAD, ST *)
FUNCTION LINEAR_BAD : INT (* Linear interpolation *)
VAR_INPUT
	PuntoMinX	: INT;
	PuntoMaxX	: INT;
	ValIn		: INT;
	PuntoMinY	: REAL;
	PuntoMaxY	: REAL;
	Decimali	: BYTE;
END_VAR
VAR
	Gain				: REAL;
	PuntoMinX_R			: REAL;
	PuntoMaxX_R			: REAL;
	Linearizzazione_R	: REAL;
END_VAR
PuntoMinX_R:=INT_TO_REAL(PuntoMinX);
PuntoMaxX_R:=INT_TO_REAL(PuntoMaxX);

Gain:=(PuntoMaxX_R-PuntoMinX_R)/(PuntoMaxY-PuntoMinY);	(* Calcolo in guadagno per la linarizzazione *)
Linearizzazione_R:=PuntoMinx+(Gain*(ValIn-PuntoMinY));	(* Ottengo il valore linearizzato *)

LINEAR_BAD:=REAL_TO_INT(Linearizzazione_R*(EXPT(10, Decimali)));  (* Ottengo intero con i decimai voluti *)
END_FUNCTION

(* POU Nodo_ETH, ST *)
PROGRAM Nodo_ETH
VAR


(* Comunizaione con nodo WAGO 192.168.100.4 *)


	Master_1				:	ETHERNET_MODBUSMASTER_UDP;
	Funktion				:	BYTE := 16#17; 				(* READ_WRITE_REGISTERS *)

	ReadAddress				:	WORD := 16#0000;			(* Startadresse 		*)
	ReadQuantity			:	WORD := 16#0005;			(* Anzahl der Worte 	*)
	Rec_Buffer				:	ARRAY[1..255] OF WORD;	(* Empfangsdaten 	*)

	WriteAddress			:	WORD := 16#0000;			(* Startadresse		*)
	WriteQuantity			:	WORD := 16#0003;			(* Anzahl der Worte	*)
	Send_Buffer			:	ARRAY[1..255] OF WORD;	(* Sendedaten			*)

	Fehler					:	WORD;
	Fertig					:	BOOL;
(*	T1						:	TON;
	Z1						:	CTU;

	WordAppoggio: WORD;   *)
	DelayAvvioCollegamentoWAGO: TON;
	DelayAggiornamento: TON;

END_VAR



VAR_INPUT
	WriteOUT: WORD;
END_VAR

VAR_OUTPUT
	ReadWord: WORD;
END_VAR
(******************************************************************************
 ****                           MAIN TASK CODE                             ****
 ******************************************************************************)

(*
WordAppoggio.0:=SPLIT07_EN;
WordAppoggio.1:=SPLIT08_EN;
WordAppoggio.2:=SPLIT09_EN;
WordAppoggio.3:=SPLIT03_EN;
WordAppoggio.4:=SPLIT02_EN;
WordAppoggio.5:=SPLIT01_EN;
WordAppoggio.6:=SPLIT06_EN;
WordAppoggio.7:=SPLIT05_EN;
WordAppoggio.8:=SPLIT04_EN;
WordAppoggio.9:=SPLIT10_EN;
WordAppoggio.10:=SPLIT11_EN;

*)


Send_Buffer[1]:=VRD04_CTRL;


Send_Buffer[3].0:=UTA01.DO_OUT;





DelayAvvioCollegamentoWAGO(IN:=TRUE , PT:=t#10s , Q=> , ET=> );
(* Provo a ritardare la lettura del nodo per veririfcare se il download del programma è più veloce *)
DelayAggiornamento(IN:=NOT DelayAggiornamento.Q,pt:=t#1s);

Fertig:=DelayAvvioCollegamentoWAGO.Q AND DelayAggiornamento.Q;

NodoWAGO();


T_S08:=Rec_Buffer[1];
T_S09:=Rec_Buffer[2];
VRD04_ST:=Rec_Buffer[3];
(*_S09:=Rec_Buffer[4];*)


UTA01_ST:=Rec_Buffer[5].0;
UTA01_AL:=Rec_Buffer[5].1;
UTA01_Antigelo:=Rec_Buffer[5].2;
UTA01_FiltroSporco:=Rec_Buffer[5].3;
UTA01_ManAut:=Rec_Buffer[5].4;
END_PROGRAM
ACTION NodoWAGO:
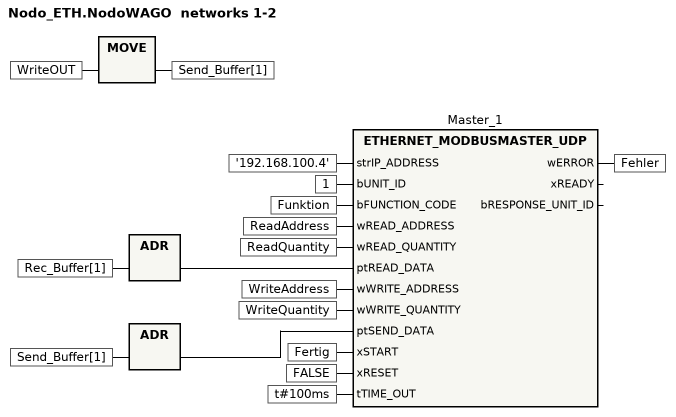
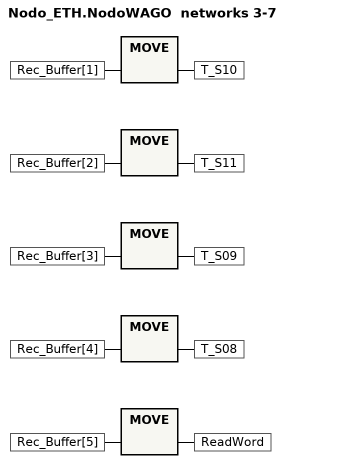
_FBD_ (* Function Block Diagram *)
NETWORK 1
	MOVE(WriteOUT) => Send_Buffer[1]
NETWORK 2
	Master_1:ETHERNET_MODBUSMASTER_UDP(strIP_ADDRESS: '192.168.100.4', bUNIT_ID: 1, bFUNCTION_CODE: Funktion, wREAD_ADDRESS: ReadAddress, wREAD_QUANTITY: ReadQuantity, ptREAD_DATA: ADR(Rec_Buffer[1]), wWRITE_ADDRESS: WriteAddress, wWRITE_QUANTITY: WriteQuantity, ptSEND_DATA: ADR(Send_Buffer[1]), xSTART: Fertig, xRESET: FALSE, tTIME_OUT: t#100ms) => Fehler
NETWORK 3
	MOVE(Rec_Buffer[1]) => T_S10
NETWORK 4
	MOVE(Rec_Buffer[2]) => T_S11
NETWORK 5
	MOVE(Rec_Buffer[3]) => T_S09
NETWORK 6
	MOVE(Rec_Buffer[4]) => T_S08
NETWORK 7
	MOVE(Rec_Buffer[5]) => ReadWord
_END_FBD_
(* the same logic as Structured Text *)
(* Network 1 *)
Send_Buffer[1] := WriteOUT;
(* Network 2 *)
Master_1(strIP_ADDRESS := '192.168.100.4', bUNIT_ID := 1, bFUNCTION_CODE := Funktion, wREAD_ADDRESS := ReadAddress, wREAD_QUANTITY := ReadQuantity, ptREAD_DATA := ADR(Rec_Buffer[1]), wWRITE_ADDRESS := WriteAddress, wWRITE_QUANTITY := WriteQuantity, ptSEND_DATA := ADR(Send_Buffer[1]), xSTART := Fertig, xRESET := FALSE, tTIME_OUT := t#100ms);
Fehler := Master_1.wERROR;
(* Network 3 *)
T_S10 := Rec_Buffer[1];
(* Network 4 *)
T_S11 := Rec_Buffer[2];
(* Network 5 *)
T_S09 := Rec_Buffer[3];
(* Network 6 *)
T_S08 := Rec_Buffer[4];
(* Network 7 *)
ReadWord := Rec_Buffer[5];
END_ACTION

(* POU Plant/SYS_Proc, ST *)
PROGRAM SYS_Proc
VAR
	fALARM_PB		:FLT_TAP;
	fALARM_TB		:FLT_TAP;
	fALARM_PM		:FLT_TAP;
	fALARM_ALARM_PM_PB_TB		:FLT_TAP;

(*	fGZB_ST			:FLT_TAP;  (* GATEWAY ZIGBEE *)*)
	fVPN_ST1		:FLT_TAP;  (* VPN CONNECT *)
	fVPN_ST2		:FLT_TAP;  (* VPN STATUS *)
	fKEY_CT_ST		:FLT_TAP;  (* DOOR1 *)
	fKEY_SCT_ST		:FLT_TAP;  (* DOOR2 *)
	fKEY_QE_ST		:FLT_TAP;  (* DOOR3 *)


	fBostAttivo	:FLT_TAP;

	fALARM_MancatoRaggiungimentoAcqua		:FLT_TAP;
	DelayfALARM_MancatoRaggiungimentoAcqua:TON;

END_VAR
(*************** ISPESL *****************)
(*
fALARM_PB(IN:=ALARM_PB);
IF fALARM_PB.EVH THEN
	LogEv(EL_AlarmStop,EO_PBV,1,1,'Over_Pressure_Alarm');
END_IF

fALARM_TB(IN:=ALARM_TB);
IF fALARM_TB.EVH THEN
	LogEv(EL_AlarmStop,EO_TBV,1,1,'Over_Temperature_Alarm');
END_IF

fALARM_PM(IN:=ALARM_PM);
IF fALARM_PM.EVH THEN
	LogEv(EL_AlarmStop,EO_PMV,1,1,'Under_Pressure_Alarm');
END_IF
*)
fALARM_ALARM_PM_PB_TB(IN:=ALARM_PM_PB_TB);
IF fALARM_ALARM_PM_PB_TB.EVH THEN
	LogEv(EL_AlarmStop,EO_PMV,1,1,'Allarmi_ISPESL');
END_IF






(****************************************)

(*### VPN Connection Check ###*)
fVPN_ST1(IN:=VPN_ST1);
IF fVPN_ST1.EVH THEN
	LogEv(EL_Log,EO_VPN,1,1,'CONNECT_ON');
END_IF
IF fVPN_ST1.EVL THEN
	LogEv(EL_Log,EO_VPN,1,2,'CONNECT_OFF');
END_IF
(*
(*### VPN Status Check ###*)
fVPN_ST2(IN:=VPN_ST2);
IF fVPN_ST2.EVH THEN
	LogEv(EL_Log,EO_VPN,1,3,'STATUS_UP');
END_IF
IF fVPN_ST2.EVL THEN
	LogEv(EL_Wrn,EO_VPN,1,4,'STATUS_DOWN');
END_IF

(*### DOOR01 Status Check ###*)
fKEY_CT_ST(IN:=KEY_CT_ST);
IF fKEY_CT_ST.EVH THEN
	LogEv(EL_Log,EO_DOOR,1,2,'Centrale_termica_Close');
END_IF
IF fKEY_CT_ST.EVL THEN
	LogEv(EL_Wrn,EO_DOOR,1,1,'Centrale_termica_Open');
END_IF

(*### DOOR02 Status Check ###*)
fKEY_SCT_ST(IN:=KEY_SCT_ST);
IF fKEY_SCT_ST.EVH THEN
	LogEv(EL_Log,EO_DOOR,2,2,'Sottocentrale_termica_Close');
END_IF
IF fKEY_SCT_ST.EVL THEN
	LogEv(EL_Wrn,EO_DOOR,2,1,'Sottocentrale_termica_Open');
END_IF
*)
(*### DOOR03 Status Check ###*)
fKEY_QE_ST(IN:=KEY_QE_ST);
IF fKEY_QE_ST.EVH THEN
	LogEv(EL_Log,EO_DOOR,3,2,'Quadro_Close');
END_IF
IF fKEY_QE_ST.EVL THEN
	LogEv(EL_Wrn,EO_DOOR,3,1,'Quadro_Open');
END_IF





(* ##### Allarme mancata Raggiungimento temperatura su mandata Acqua ####### *)


DelayfALARM_MancatoRaggiungimentoAcqua(IN:=(CAL01.Run),PT:=DINT_TO_TIME(DelayAllarmeTemperaturaNonRaggiunta*60000));

 (* in questo caso il delta viene applicato al Set point fisico che si da alla caldaia *)

fALARM_MancatoRaggiungimentoAcqua(IN:=DelayfALARM_MancatoRaggiungimentoAcqua.Q
									AND ( TPV02.AVG < CAL01.SetPoint -  DeltaInterventoAllarmeTempeaturaNonRaggiuta));
IF fALARM_MancatoRaggiungimentoAcqua.EVH THEN
	LogEv(EL_AlarmStop,EO_SYS,0,11,'Mancato_Raggiungimento_Temp');
END_IF

(* Segnalazione Boost Attivo *)

fBostAttivo(IN:=BitAbilitaBoost AND (THER250.SetPoint>TPV08.AVG));
IF fBostAttivo.EVH THEN
	LogEv(EL_Log,EO_SYS,0,14,'Boost_Attivo');
END_IF
IF fBostAttivo.EVL THEN
	LogEv(EL_Log,EO_SYS,0,15,'Boost_Non_Attivo');
END_IF
END_PROGRAM

(* POU Utils Functions/AVERAGE_T, ST *)
FUNCTION_BLOCK AVERAGE_T
VAR_INPUT
	IN: 	INT;
END_VAR
VAR_OUTPUT
	HI:		INT;
	AVG:	INT;
	LOW:	INT;
	ERR:	BOOL;
END_VAR
VAR
	sum:	DINT;
	cnt:	WORD;
END_VAR
IF cnt>=65000 THEN
	ERR:=TRUE;
	Read();
	sum := sum - AVG;
	cnt := cnt + 1;
END_IF

sum := sum + IN;
cnt := cnt + 1;

IF IN<LOW THEN  LOW:=IN; END_IF
IF IN>HI  THEN HI :=IN; END_IF
END_FUNCTION_BLOCK
ACTION Read:
AVG := DINT_TO_INT(sum/cnt);
END_ACTION
ACTION Reset:
HI:=IN;
AVG:=IN;
LOW:=IN;
ERR:=FALSE;

sum:=IN;
cnt:=1;
END_ACTION

(* POU Utils/CSV_Log, ST *)
FUNCTION CSV_Log : BOOL
VAR_INPUT
END_VAR
VAR CONSTANT
	LogFileName:STRING:='S:\LOGS_ID1V3.CSV';
END_VAR
VAR
	s1 : STRING(180);
	hFile: 	DWORD;
END_VAR
(* Check file presence *)
hFile:=SysFileOpen(LogFileName,'r');
IF hFile=0 THEN
	(*** File not exist *** Create file and write header *)
	hFile:=SysFileOpen(LogFileName,'w');
	IF hFile<>0 THEN
		(* Write CSV header *)
		s1:='DATE-TIME;T-Amb;T-S02;T-S03;T-S04;T-S05;T-S06;T-S07;T-S08;T-S09;';
		SysFileWrite(hFile, ADR(s1), LEN(s1));
		s1:='T-VRD01-AvgSend;T-VRD02-AvgSendT-VRD01-AvgSend;';
		SysFileWrite(hFile, ADR(s1), LEN(s1));
		SysFileWrite(hFile, ADR(Logger_CRLF), LEN(Logger_CRLF));
	END_IF
ELSE
	(*** File exist *** Close file and reopen in append mode *)
	SysFileClose(hFile);
	hFile:=SysFileOpen(LogFileName,'a');
END_IF

(* Log to file *)
IF hFile<>0 THEN
	(* Date stamp *)
	s1:=REPLACE( Sys.Time_LogString , ' ' , 1 , 11 );
	SysFileWrite(hFile, ADR(s1), LEN(s1));
	(* Log data *)
	s1:=CONCAT(';', INT_TO_STRING(TPV01.IN) );
	s1:=CONCAT(s1 , ';' );
	s1:=CONCAT(s1 , INT_TO_STRING(TPV02.IN) );
	s1:=CONCAT(s1 , ';' );
	s1:=CONCAT(s1 , INT_TO_STRING(TPV03.IN) );
	s1:=CONCAT(s1 , ';' );
	s1:=CONCAT(s1 , INT_TO_STRING(TPV04.IN) );
	s1:=CONCAT(s1 , ';' );
	s1:=CONCAT(s1 , INT_TO_STRING(TPV05.IN) );
	s1:=CONCAT(s1 , ';' );
	s1:=CONCAT(s1 , INT_TO_STRING(TPV06.IN) );
	s1:=CONCAT(s1 , ';' );
	s1:=CONCAT(s1 , INT_TO_STRING(TPV07.IN) );
	s1:=CONCAT(s1 , ';' );
	s1:=CONCAT(s1 , INT_TO_STRING(TPV08.IN) );
	s1:=CONCAT(s1 , ';' );
	s1:=CONCAT(s1 , INT_TO_STRING(TPV09.IN) );
	s1:=CONCAT(s1 , ';' );

	VRD01.Log_AvgTemp.Read();
	VRD02.Log_AvgTemp.Read();
(* VRD03 Esclusa perchè bypassata *)
(*	VRD03.Log_AvgTemp.Read();*)

	s1:=CONCAT(s1 , INT_TO_STRING(VRD01.Log_AvgTemp.AVG) );
	s1:=CONCAT(s1 , ';' );
	s1:=CONCAT(s1 , INT_TO_STRING(VRD02.Log_AvgTemp.AVG) );
	s1:=CONCAT(s1 , ';' );
(* VRD03 Esclusa perchè bypassata *)
(*	s1:=CONCAT(s1 , INT_TO_STRING(VRD03.Log_AvgTemp.AVG) );
	s1:=CONCAT(s1 , ';' ); *)
	VRD01.Log_AvgTemp.Reset();
	VRD02.Log_AvgTemp.Reset();
(* VRD03 Esclusa perchè bypassata *)
(*	VRD03.Log_AvgTemp.Reset();*)
	SysFileWrite(hFile, ADR(s1), LEN(s1));
	(* Add line CRLF and close *)
	SysFileWrite(hFile, ADR(Logger_CRLF), LEN(Logger_CRLF));
	SysFileClose(hFile);
END_IF
END_FUNCTION

(* POU Utils Functions/FLT_EVENT, ST *)
FUNCTION_BLOCK FLT_EVENT
VAR_INPUT
	IN		: BOOL;
	INITEV	: BOOL:=TRUE;
END_VAR
VAR_OUTPUT
	EVH		: BOOL;
	EVL		: BOOL;
END_VAR
VAR
	init	: BOOL:=FALSE;
	old		: BOOL;
END_VAR
EVH:=FALSE;
EVL:=FALSE;

IF NOT init THEN
	init:=TRUE;
	IF INITEV THEN
		old := NOT IN;
	ELSE
		old := IN;
	END_IF
END_IF

IF old<>IN THEN
	old:=IN;
	IF IN THEN EVH:=TRUE; ELSE EVL:=TRUE; END_IF
END_IF
END_FUNCTION_BLOCK

(* POU Utils Functions/FLT_TIME, ST *)
FUNCTION_BLOCK FLT_TIME
VAR_INPUT
	IN		: BOOL;
	TTAP	: TIME:=T#5s;
	INITEV	: BOOL:=TRUE;
END_VAR
VAR_OUTPUT
	OUT		: BOOL;
	EVH		: BOOL;
	EVL		: BOOL;
END_VAR
VAR
	init	: BOOL:=FALSE;
	timer	: TON;
END_VAR
EVH:=FALSE;
EVL:=FALSE;

IF NOT init THEN
	init := TRUE;
	IF INITEV THEN
		OUT  := NOT IN;
	ELSE
		OUT  := IN;
	END_IF
END_IF

IF OUT<>IN THEN
	timer(IN:=TRUE,PT:=TTAP);
	IF timer.Q THEN
		OUT:=IN;
		timer(IN:=FALSE);
		IF OUT THEN EVH:=TRUE; ELSE EVL:=TRUE; END_IF
	END_IF
ELSE
	timer(IN:=FALSE);
END_IF
END_FUNCTION_BLOCK

(* POU Utils Functions/LAMP_AL_GENERALE, ST *)
FUNCTION_BLOCK LAMP_AL_GENERALE
VAR_INPUT

	Allarme: BOOL;
	Warning: BOOL;
END_VAR
VAR_OUTPUT
	SistemaOK:BOOL;
	SistemaInAllarme:BOOL;
	SistemaWarning:BOOL;
	AllarmeLampada:BOOL;
END_VAR
VAR
	Lampeggio:BLINK;
END_VAR
IF Allarme THEN       					(* Se Allarme Attivo Lucde fissa ON *)
	SistemaInAllarme:=TRUE;
	SistemaWarning:=FALSE;
	AllarmeLampada:=TRUE;
ELSIF Warning THEN					(* Se Allarme Attivo Lucde fissa pulse *)
	SistemaInAllarme:=FALSE;
	SistemaWarning:=TRUE;
	Lampeggio(ENABLE:=TRUE , TIMELOW:=t#1s , TIMEHIGH:=t#1s , OUT=>AllarmeLampada );
ELSE
	SistemaInAllarme:=FALSE;
	SistemaWarning:=FALSE;
	AllarmeLampada:=FALSE;
END_IF
END_FUNCTION_BLOCK

